C07280=1058.171,437.212,373.375,176.008,40.727,157.978
C07281=1058.182,437.458,373.325,176.019,40.739,157.981
C07282=1058.192,437.701,373.276,176.030,40.751,157.985
C07283=1058.202,437.947,373.225,176.042,40.763,157.989
C07284=1058.213,438.192,373.176,176.053,40.775,157.993
C07285=1058.223,438.436,373.126,176.064,40.788,157.997
C07286=1058.234,438.681,373.077,176.075,40.799,158.000
C07287=1058.244,438.926,373.026,176.086,40.811,158.004
C07288=1058.254,439.170,372.977,176.098,40.824,158.008
C07289=1058.265,439.415,372.926,176.109,40.836,158.012
C07290=1058.276,439.660,372.877,176.121,40.848,158.016
C07291=1058.286,439.904,372.826,176.133,40.860,158.020
C07292=1058.296,440.149,372.776,176.144,40.873,158.024
C07293=1058.307,440.394,372.725,176.155,40.885,158.028
C07294=1058.317,440.638,372.675,176.167,40.897,158.032
C07295=1058.328,440.882,372.625,176.179,40.909,158.035
C07296=1058.338,441.128,372.575,176.191,40.922,158.040
C07297=1058.349,441.372,372.525,176.202,40.935,158.044
C07298=1058.359,441.617,372.474,176.215,40.947,158.048
C07299=1058.370,441.861,372.423,176.226,40.960,158.052
C07300=1058.381,442.106,372.373,176.238,40.973,158.056
C07301=1058.391,442.350,372.322,176.250,40.985,158.060
C07302=1058.402,442.595,372.272,176.262,40.997,158.064
C07303=1058.414,442.840,372.220,176.274,41.010,158.068
C07304=1058.424,443.084,372.169,176.286,41.023,158.072
C07305=1058.435,443.329,372.118,176.299,41.036,158.076
C07306=1058.446,443.573,372.067,176.311,41.049,158.080
C07307=1058.456,443.817,372.017,176.323,41.062,158.085
C07308=1058.467,444.062,371.965,176.335,41.075,158.089
C07309=1058.479,444.330,371.909,176.349,41.089,158.094
C07310=1058.491,444.598,371.853,176.363,41.103,158.098
C07311=1058.503,444.866,371.797,176.377,41.117,158.103
C07312=1058.515,445.134,371.741,176.390,41.132,158.108
C07313=1058.525,445.378,371.690,176.403,41.145,158.112
C07314=1058.537,445.622,371.638,176.415,41.158,158.116
C07315=1058.548,445.867,371.587,176.428,41.171,158.121
C07316=1058.559,446.111,371.535,176.441,41.185,158.125
C07317=1058.570,446.355,371.484,176.454,41.198,158.129
C07318=1058.582,446.599,371.432,176.467,41.211,158.134
C07319=1058.592,446.842,371.380,176.480,41.225,158.138
C07320=1058.604,447.087,371.329,176.493,41.238,158.143
C07321=1058.616,447.330,371.279,176.506,41.251,158.147
C07322=1058.629,447.573,371.228,176.519,41.264,158.151
C07323=1058.642,447.817,371.178,176.532,41.277,158.156
C07324=1058.658,448.062,371.130,176.546,41.289,158.160
C07325=1058.673,448.306,371.080,176.558,41.302,158.164
C07326=1058.690,448.550,371.033,176.572,41.314,158.168
C07327=1058.707,448.795,370.986,176.586,41.325,158.172
C07328=1058.725,449.040,370.938,176.599,41.337,158.176
C07329=1058.744,449.285,370.893,176.613,41.348,158.180
C07330=1058.764,449.530,370.848,176.626,41.360,158.184
C07331=1058.785,449.776,370.802,176.641,41.371,158.188
C07332=1058.806,450.022,370.758,176.654,41.381,158.192
C07333=1058.477,450.035,370.476,176.650,41.491,158.222
C07334=1058.456,449.789,370.520,176.636,41.480,158.218
C07335=1058.436,449.544,370.565,176.622,41.470,158.214
C07336=1058.416,449.299,370.610,176.608,41.459,158.210
C07337=1058.396,449.054,370.656,176.594,41.447,158.206
C07338=1058.378,448.810,370.703,176.581,41.436,158.202
C07339=1058.361,448.565,370.750,176.567,41.424,158.198
C07340=1058.344,448.320,370.798,176.553,41.412,158.194
C07341=1058.328,448.076,370.847,176.540,41.400,158.190
C07342=1058.313,447.831,370.896,176.527,41.387,158.186
C07343=1058.299,447.587,370.945,176.514,41.375,158.182
C07344=1058.286,447.343,370.995,176.501,41.362,158.177
C07345=1058.273,447.100,371.046,176.487,41.349,158.173
C07346=1058.262,446.857,371.097,176.474,41.336,158.169
C07347=1058.251,446.613,371.149,176.461,41.322,158.164
C07348=1058.239,446.369,371.201,176.448,41.309,158.160
C07349=1058.229,446.124,371.252,176.435,41.295,158.155
C07350=1058.218,445.881,371.303,176.422,41.282,158.151
C07351=1058.206,445.636,371.355,176.409,41.269,158.147
C07352=1058.195,445.392,371.407,176.396,41.256,158.142
C07353=1058.184,445.147,371.459,176.384,41.243,158.138
C07354=1058.173,444.899,371.510,176.371,41.230,158.134
C07355=1058.162,444.651,371.563,176.359,41.217,158.129
C07356=1058.151,444.401,371.615,176.346,41.204,158.125
C07357=1058.139,444.153,371.667,176.333,41.190,158.121
C07358=1058.129,443.908,371.718,176.321,41.177,158.116
C07359=1058.117,443.664,371.769,176.308,41.164,158.112
C07360=1058.107,443.419,371.820,176.296,41.151,158.108
C07361=1058.096,443.175,371.872,176.283,41.139,158.104
C07362=1058.085,442.930,371.922,176.271,41.126,158.099
C07363=1058.075,442.686,371.974,176.259,41.113,158.095
C07364=1058.064,442.442,372.024,176.246,41.101,158.091
C07365=1058.054,442.197,372.075,176.235,41.088,158.087
C07366=1058.042,441.952,372.126,176.223,41.075,158.083
C07367=1058.031,441.707,372.176,176.211,41.063,158.079
C07368=1058.021,441.463,372.227,176.199,41.050,158.075
C07369=1058.010,441.218,372.277,176.186,41.038,158.071
C07370=1058.000,440.974,372.328,176.175,41.026,158.067
C07371=1057.989,440.729,372.379,176.163,41.013,158.063
C07372=1057.978,440.485,372.429,176.151,41.001,158.059
C07373=1057.968,440.240,372.479,176.139,40.988,158.055
C07374=1057.957,439.996,372.529,176.128,40.976,158.051
C07375=1057.947,439.751,372.579,176.117,40.964,158.047
C07376=1057.937,439.506,372.630,176.105,40.952,158.043
C07377=1057.926,439.261,372.680,176.093,40.940,158.039
C07378=1057.915,439.016,372.730,176.082,40.928,158.035
C07379=1057.905,438.772,372.780,176.070,40.915,158.031
C07380=1057.895,438.527,372.830,176.059,40.904,158.028
C07381=1057.884,438.282,372.879,176.048,40.892,158.024
C07382=1057.874,438.038,372.929,176.036,40.879,158.020
C07383=1057.864,437.793,372.980,176.025,40.867,158.016
C07384=1057.853,437.548,373.029,176.014,40.855,158.012
C07385=1057.843,437.304,373.078,176.003,40.844,158.009
C07386=1057.832,437.059,373.128,175.992,40.832,158.005
C07387=1057.822,436.814,373.178,175.981,40.820,158.001
C07388=1057.812,436.569,373.227,175.970,40.808,157.997
C07389=1057.801,436.324,373.276,175.959,40.797,157.994
C07390=1057.790,436.079,373.326,175.947,40.785,157.990
C07391=1057.780,435.834,373.375,175.936,40.774,157.986
C07392=1057.770,435.589,373.424,175.925,40.762,157.983
C07393=1057.760,435.345,373.473,175.915,40.751,157.979
C07394=1057.749,435.100,373.523,175.903,40.739,157.975
C07395=1057.739,434.855,373.572,175.893,40.727,157.972
C07396=1057.729,434.610,373.621,175.882,40.716,157.968
C07397=1057.719,434.365,373.670,175.872,40.705,157.965
C07398=1057.709,434.120,373.719,175.861,40.694,157.961
C07399=1057.699,433.875,373.767,175.851,40.682,157.958
C07400=1057.689,433.630,373.816,175.840,40.671,157.954
C07401=1057.679,433.385,373.866,175.829,40.660,157.951
C07402=1057.669,433.140,373.914,175.819,40.648,157.947
C07403=1057.658,432.895,373.963,175.809,40.637,157.944
C07404=1057.649,432.650,374.012,175.798,40.626,157.940
C07405=1057.639,432.405,374.061,175.788,40.615,157.937
C07406=1057.629,432.160,374.109,175.777,40.604,157.933
C07407=1057.619,431.915,374.158,175.767,40.593,157.930
C07408=1057.609,431.670,374.206,175.757,40.582,157.926
C07409=1057.600,431.425,374.255,175.746,40.571,157.923
C07410=1057.585,431.059,374.327,175.732,40.554,157.918
C07411=1057.571,430.692,374.399,175.716,40.538,157.913
C07412=1057.556,430.326,374.472,175.701,40.521,157.908
C07413=1057.541,429.960,374.544,175.686,40.505,157.903
C07414=1057.531,429.714,374.591,175.676,40.495,157.900
C07415=1057.522,429.469,374.640,175.666,40.484,157.896
C07416=1057.512,429.224,374.687,175.657,40.473,157.893
C07417=1057.502,428.979,374.736,175.646,40.462,157.890
C07418=1057.492,428.734,374.783,175.637,40.452,157.886
C07419=1057.482,428.489,374.831,175.627,40.441,157.883
C07420=1057.472,428.243,374.879,175.617,40.431,157.880
C07421=1057.463,427.998,374.927,175.607,40.420,157.877
C07422=1057.453,427.753,374.974,175.598,40.409,157.873
C07423=1057.444,427.508,375.022,175.587,40.399,157.870
C07424=1057.434,427.263,375.070,175.578,40.388,157.867
C07425=1057.424,427.017,375.117,175.569,40.378,157.864
C07426=1057.415,426.772,375.165,175.559,40.368,157.861
C07427=1057.406,426.527,375.213,175.550,40.357,157.858
C07428=1057.395,426.282,375.260,175.540,40.347,157.854
C07429=1057.386,426.036,375.308,175.530,40.337,157.851
C07430=1057.376,425.791,375.354,175.521,40.327,157.848
C07431=1057.367,425.545,375.402,175.512,40.316,157.845
C07432=1057.357,425.300,375.449,175.503,40.306,157.842
C07433=1057.348,425.055,375.496,175.493,40.296,157.839
C07434=1057.338,424.810,375.543,175.484,40.285,157.836
C07435=1057.329,424.564,375.590,175.475,40.276,157.833
C07436=1057.319,424.319,375.637,175.466,40.266,157.830
C07437=1057.309,424.073,375.684,175.457,40.256,157.827
C07438=1057.301,423.828,375.731,175.446,40.245,157.824
C07439=1057.291,423.582,375.778,175.437,40.236,157.821
C07440=1057.282,423.337,375.825,175.429,40.226,157.818
C07441=1057.272,423.091,375.872,175.420,40.215,157.815
C07442=1057.262,422.847,375.919,175.411,40.206,157.812
C07443=1057.254,422.601,375.965,175.402,40.196,157.809
C07444=1057.244,422.355,376.012,175.393,40.186,157.806
C07445=1057.235,422.110,376.059,175.384,40.176,157.803
C07446=1057.225,421.865,376.106,175.375,40.167,157.800
C07447=1057.216,421.619,376.152,175.365,40.156,157.797
C07448=1057.207,421.374,376.199,175.356,40.147,157.794
C07449=1057.197,421.128,376.245,175.347,40.137,157.791
C07450=1057.188,420.883,376.291,175.339,40.127,157.788
C07451=1057.180,420.637,376.338,175.330,40.117,157.785
C07452=1057.170,420.392,376.384,175.321,40.108,157.783
C07453=1057.161,420.146,376.431,175.313,40.099,157.780
C07454=1057.152,419.901,376.477,175.304,40.089,157.777
C07455=1057.143,419.655,376.523,175.296,40.079,157.774
C07456=1057.134,419.410,376.569,175.287,40.070,157.771
C07457=1057.124,419.164,376.615,175.278,40.060,157.768
C07458=1057.115,418.918,376.661,175.270,40.051,157.766
C07459=1057.105,418.673,376.707,175.261,40.041,157.763
C07460=1057.097,418.427,376.754,175.252,40.032,157.760
C07461=1057.088,418.181,376.799,175.243,40.023,157.757
C07462=1057.079,417.936,376.845,175.236,40.014,157.755
C07463=1057.070,417.690,376.891,175.227,40.004,157.752
C07464=1057.060,417.445,376.937,175.218,39.995,157.749
C07465=1057.051,417.199,376.983,175.210,39.985,157.746
C07466=1057.039,416.854,377.046,175.198,39.973,157.743
C07467=1057.025,416.509,377.111,175.186,39.960,157.739
C07468=1057.013,416.164,377.175,175.175,39.947,157.735
C07469=1057.001,415.819,377.239,175.164,39.934,157.731
C07470=1056.992,415.573,377.284,175.155,39.925,157.729
C07471=1056.983,415.327,377.330,175.147,39.916,157.726
C07472=1056.974,415.081,377.375,175.139,39.907,157.723
C07473=1056.965,414.836,377.420,175.131,39.897,157.721
C07474=1056.956,414.591,377.466,175.122,39.889,157.718
C07475=1056.947,414.345,377.511,175.115,39.880,157.716
C07476=1056.938,414.099,377.556,175.106,39.871,157.713
C07477=1056.929,413.853,377.602,175.098,39.862,157.710
C07478=1056.921,413.608,377.647,175.090,39.853,157.708
C07479=1056.912,413.362,377.692,175.082,39.844,157.705
C07480=1056.902,413.117,377.737,175.075,39.835,157.702
C07481=1056.894,412.870,377.782,175.066,39.826,157.700
C07482=1056.885,412.624,377.827,175.058,39.817,157.697
C07483=1056.876,412.378,377.872,175.050,39.809,157.695
C07484=1056.867,412.133,377.916,175.042,39.800,157.692
C07485=1056.858,411.887,377.962,175.035,39.791,157.690
C07486=1056.849,411.641,378.007,175.026,39.783,157.687
C07487=1056.840,411.396,378.051,175.019,39.774,157.685
C07488=1056.832,411.150,378.096,175.011,39.766,157.682
C07489=1056.823,410.903,378.140,175.004,39.757,157.680
C07490=1056.814,410.658,378.185,174.995,39.749,157.677
C07491=1056.805,410.412,378.230,174.988,39.740,157.675
C07492=1056.797,410.166,378.274,174.981,39.731,157.673
C07493=1056.787,409.921,378.319,174.973,39.723,157.670
C07494=1056.779,409.674,378.363,174.965,39.714,157.668
C07495=1056.771,409.428,378.408,174.957,39.705,157.665
C07496=1056.761,409.182,378.452,174.950,39.697,157.663
C07497=1056.753,408.936,378.496,174.942,39.689,157.660
C07498=1056.745,408.691,378.541,174.935,39.680,157.658
C07499=1056.735,408.445,378.585,174.927,39.672,157.656
C07500=1056.727,408.199,378.630,174.919,39.663,157.653
C07501=1056.719,407.953,378.674,174.912,39.655,157.651
C07502=1056.710,407.708,378.718,174.905,39.647,157.648
C07503=1056.702,407.462,378.763,174.897,39.638,157.646
C07504=1056.693,407.215,378.807,174.890,39.630,157.644
C07505=1056.685,406.969,378.850,174.883,39.622,157.641
C07506=1056.676,406.724,378.895,174.875,39.614,157.639
C07507=1056.667,406.477,378.939,174.868,39.605,157.637
C07508=1056.659,406.232,378.983,174.860,39.597,157.634
C07509=1056.651,405.986,379.027,174.852,39.589,157.632
C07510=1056.642,405.739,379.071,174.845,39.581,157.630
C07511=1056.634,405.493,379.115,174.838,39.573,157.627
C07512=1056.625,405.248,379.159,174.831,39.565,157.625
C07513=1056.617,405.002,379.202,174.823,39.556,157.623
C07514=1056.608,404.756,379.246,174.816,39.549,157.620
C07515=1056.600,404.509,379.290,174.809,39.540,157.618
C07516=1056.591,404.264,379.334,174.802,39.532,157.616
C07517=1056.583,404.018,379.377,174.794,39.525,157.614
C07518=1056.575,403.772,379.421,174.787,39.517,157.611
C07519=1056.566,403.526,379.464,174.781,39.508,157.609
C07520=1056.558,403.280,379.508,174.774,39.500,157.607
C07521=1056.550,403.034,379.552,174.767,39.493,157.605
C07522=1056.538,402.694,379.611,174.757,39.482,157.602
C07523=1056.526,402.355,379.671,174.747,39.471,157.599
C07524=1056.515,402.016,379.731,174.737,39.460,157.596
C07525=1056.503,401.678,379.791,174.728,39.450,157.593
C07526=1056.495,401.431,379.834,174.721,39.442,157.590
C07527=1056.487,401.185,379.877,174.714,39.434,157.588
C07528=1056.478,400.939,379.920,174.707,39.426,157.586
C07529=1056.470,400.693,379.963,174.700,39.419,157.584
C07530=1056.461,400.447,380.006,174.693,39.411,157.582
C07531=1056.453,400.201,380.049,174.687,39.403,157.580
C07532=1056.445,399.954,380.092,174.679,39.396,157.578
C07533=1056.437,399.708,380.135,174.672,39.388,157.575
C07534=1056.428,399.462,380.178,174.665,39.380,157.573
C07535=1056.420,399.216,380.221,174.658,39.373,157.571
C07536=1056.411,398.970,380.264,174.652,39.365,157.569
C07537=1056.403,398.724,380.307,174.645,39.358,157.567
C07538=1056.395,398.478,380.349,174.638,39.350,157.565
C07539=1056.387,398.232,380.392,174.631,39.342,157.563
C07540=1056.379,397.985,380.436,174.625,39.335,157.561
C07541=1056.371,397.739,380.478,174.618,39.328,157.559
C07542=1056.363,397.493,380.521,174.611,39.320,157.557
C07543=1056.355,397.247,380.563,174.605,39.313,157.555
C07544=1056.346,397.001,380.606,174.599,39.306,157.553
C07545=1056.339,396.755,380.648,174.592,39.298,157.550
C07546=1056.330,396.509,380.691,174.585,39.291,157.548
C07547=1056.322,396.262,380.734,174.579,39.283,157.546
C07548=1056.313,396.016,380.777,174.572,39.276,157.544
C07549=1056.305,395.770,380.818,174.565,39.269,157.542
C07550=1056.297,395.523,380.860,174.559,39.261,157.540
C07551=1056.288,395.277,380.903,174.552,39.254,157.538
C07552=1056.281,395.031,380.945,174.545,39.247,157.536
C07553=1056.272,394.785,380.988,174.539,39.239,157.534
C07554=1056.265,394.539,381.029,174.532,39.232,157.532
C07555=1056.256,394.293,381.072,174.527,39.225,157.530
C07556=1056.249,394.047,381.114,174.520,39.218,157.528
C07557=1056.241,393.800,381.157,174.513,39.211,157.526
C07558=1056.232,393.554,381.198,174.507,39.204,157.524
C07559=1056.224,393.308,381.240,174.500,39.197,157.523
C07560=1056.216,393.062,381.282,174.494,39.189,157.520
C07561=1056.208,392.815,381.325,174.487,39.182,157.519
C07562=1056.201,392.569,381.367,174.481,39.175,157.517
C07563=1056.192,392.323,381.408,174.475,39.168,157.515
C07564=1056.184,392.077,381.450,174.468,39.161,157.513
C07565=1056.176,391.830,381.493,174.462,39.154,157.511
C07566=1056.168,391.584,381.535,174.455,39.147,157.509
C07567=1056.160,391.338,381.576,174.450,39.140,157.507
C07568=1056.152,391.091,381.617,174.443,39.133,157.505
C07569=1056.145,390.845,381.659,174.437,39.126,157.503
C07570=1056.136,390.599,381.701,174.430,39.119,157.501
C07571=1056.128,390.353,381.743,174.425,39.112,157.499
C07572=1056.121,390.106,381.784,174.418,39.105,157.498
C07573=1056.112,389.861,381.826,174.412,39.098,157.496
C07574=1056.104,389.614,381.868,174.405,39.092,157.494
C07575=1056.097,389.367,381.909,174.400,39.085,157.492
C07576=1056.088,389.121,381.951,174.393,39.078,157.490
C07577=1056.080,388.875,381.992,174.387,39.071,157.488
C07578=1056.070,388.553,382.046,174.379,39.062,157.486
C07579=1056.059,388.231,382.100,174.371,39.054,157.484
C07580=1056.049,387.910,382.154,174.364,39.045,157.481
C07581=1056.039,387.589,382.207,174.356,39.036,157.479
C07582=1056.030,387.342,382.248,174.349,39.029,157.477
C07583=1056.023,387.096,382.290,174.343,39.023,157.475
C07584=1056.015,386.849,382.331,174.337,39.016,157.473
C07585=1056.007,386.603,382.372,174.331,39.010,157.472
C07586=1055.999,386.357,382.413,174.325,39.003,157.470
C07587=1055.990,386.110,382.454,174.319,38.996,157.468
C07588=1055.983,385.864,382.496,174.313,38.989,157.466
C07589=1055.975,385.617,382.536,174.307,38.983,157.464
C07590=1055.968,385.371,382.578,174.301,38.977,157.463
C07591=1055.960,385.124,382.618,174.295,38.970,157.461
C07592=1055.952,384.878,382.659,174.289,38.963,157.459
C07593=1055.944,384.632,382.700,174.283,38.957,157.457
C07594=1055.936,384.385,382.741,174.277,38.950,157.456
C07595=1055.929,384.139,382.782,174.272,38.944,157.454
C07596=1055.921,383.892,382.822,174.266,38.937,157.452
C07597=1055.913,383.646,382.863,174.259,38.931,157.450
C07598=1055.906,383.400,382.904,174.254,38.924,157.449
C07599=1055.898,383.153,382.945,174.248,38.918,157.447
C07600=1055.890,382.906,382.985,174.242,38.911,157.445
C07601=1055.883,382.660,383.026,174.236,38.905,157.443
C07602=1055.875,382.413,383.067,174.231,38.898,157.442
C07603=1055.867,382.167,383.108,174.225,38.892,157.440
C07604=1055.859,381.921,383.149,174.219,38.886,157.438
C07605=1055.852,381.674,383.189,174.213,38.879,157.437
C07606=1055.844,381.427,383.230,174.208,38.873,157.435
C07607=1055.836,381.181,383.270,174.202,38.867,157.433
C07608=1055.829,380.934,383.310,174.197,38.860,157.432
C07609=1055.822,380.688,383.351,174.190,38.854,157.430
C07610=1055.814,380.441,383.391,174.184,38.847,157.428
C07611=1055.806,380.195,383.432,174.179,38.842,157.427
C07612=1055.799,379.948,383.472,174.173,38.835,157.425
C07613=1055.791,379.702,383.512,174.168,38.829,157.423
C07614=1055.783,379.455,383.552,174.162,38.823,157.422
C07615=1055.775,379.208,383.592,174.156,38.817,157.420
C07616=1055.767,378.962,383.633,174.151,38.810,157.418
C07617=1055.760,378.715,383.672,174.145,38.804,157.417
C07618=1055.752,378.468,383.712,174.140,38.798,157.415
C07619=1055.744,378.222,383.753,174.134,38.792,157.414
C07620=1055.736,377.975,383.793,174.129,38.786,157.412
C07621=1055.729,377.728,383.833,174.122,38.780,157.410
C07622=1055.722,377.482,383.872,174.117,38.774,157.409
C07623=1055.714,377.236,383.913,174.112,38.768,157.407
C07624=1055.706,376.989,383.953,174.106,38.761,157.405
C07625=1055.698,376.742,383.993,174.101,38.755,157.404
C07626=1055.691,376.496,384.032,174.095,38.750,157.402
C07627=1055.683,376.249,384.072,174.090,38.744,157.401
C07628=1055.676,376.002,384.112,174.084,38.737,157.399
C07629=1055.668,375.756,384.152,174.079,38.731,157.397
C07630=1055.661,375.509,384.192,174.074,38.725,157.396
C07631=1055.653,375.262,384.232,174.067,38.719,157.394
C07632=1055.646,375.016,384.271,174.062,38.713,157.393
C07633=1055.638,374.769,384.311,174.056,38.708,157.391
C07634=1055.630,374.479,384.357,174.051,38.700,157.389
C07635=1055.621,374.189,384.404,174.044,38.693,157.388
C07636=1055.611,373.900,384.451,174.038,38.686,157.386
C07637=1055.603,373.610,384.497,174.031,38.679,157.384
C07638=1055.596,373.363,384.537,174.026,38.673,157.382
C07639=1055.589,373.116,384.576,174.020,38.668,157.381
C07640=1055.581,372.869,384.616,174.015,38.662,157.379
C07641=1055.574,372.623,384.656,174.011,38.656,157.378
C07642=1055.567,372.376,384.695,174.005,38.650,157.376
C07643=1055.559,372.130,384.734,174.000,38.644,157.375
C07644=1055.552,371.883,384.774,173.995,38.638,157.373
C07645=1055.544,371.636,384.813,173.989,38.633,157.372
C07646=1055.536,371.389,384.853,173.984,38.627,157.370
C07647=1055.530,371.142,384.891,173.979,38.622,157.369
C07648=1055.521,370.896,384.931,173.973,38.616,157.367
C07649=1055.514,370.649,384.970,173.968,38.610,157.366
C07650=1055.506,370.402,385.009,173.963,38.604,157.364
C07651=1055.499,370.156,385.048,173.958,38.599,157.363
C07652=1055.492,369.908,385.087,173.952,38.593,157.361
C07653=1055.484,369.662,385.126,173.947,38.587,157.360
C07654=1055.476,369.415,385.165,173.942,38.581,157.358
C07655=1055.470,369.168,385.204,173.936,38.576,157.357
C07656=1055.462,368.922,385.243,173.931,38.570,157.355
C07657=1055.454,368.674,385.282,173.926,38.565,157.354
C07658=1055.447,368.428,385.320,173.921,38.559,157.353
C07659=1055.440,368.181,385.359,173.916,38.553,157.351
C07660=1055.432,367.934,385.399,173.911,38.548,157.350
C07661=1055.425,367.688,385.437,173.906,38.542,157.348
C07662=1055.418,367.441,385.476,173.901,38.537,157.347
C07663=1055.410,367.194,385.515,173.895,38.531,157.345
C07664=1055.403,366.947,385.554,173.890,38.526,157.344
C07665=1055.396,366.700,385.592,173.885,38.520,157.342
C07666=1055.389,366.474,385.628,173.881,38.515,157.341
C07667=1055.383,366.248,385.663,173.876,38.510,157.340
C07668=1055.375,366.022,385.699,173.871,38.505,157.339
C07669=1055.369,365.796,385.735,173.866,38.500,157.337
C07670=1055.362,365.570,385.770,173.862,38.494,157.336
C07671=1055.355,365.344,385.806,173.857,38.490,157.335
C07672=1055.349,365.118,385.840,173.853,38.485,157.333
C07673=1055.342,364.892,385.876,173.848,38.480,157.332
C07674=1055.335,364.645,385.914,173.843,38.474,157.331
C07675=1055.328,364.397,385.953,173.839,38.469,157.329
C07676=1055.320,364.151,385.991,173.833,38.463,157.328
C07677=1055.313,363.904,386.030,173.828,38.458,157.326
C07678=1055.306,363.657,386.068,173.823,38.453,157.325
C07679=1055.299,363.411,386.107,173.819,38.447,157.324
C07680=1055.292,363.163,386.145,173.814,38.442,157.322
C07681=1055.284,362.916,386.183,173.808,38.436,157.321
C07682=1055.277,362.669,386.222,173.803,38.431,157.320
C07683=1055.270,362.422,386.260,173.798,38.426,157.318
C07684=1055.262,362.176,386.298,173.794,38.420,157.317
C07685=1055.256,361.928,386.336,173.789,38.415,157.315
C07686=1055.248,361.682,386.374,173.784,38.410,157.314
C07687=1055.241,361.435,386.412,173.779,38.405,157.313
C07688=1055.234,361.188,386.451,173.774,38.399,157.311
C07689=1055.226,360.941,386.489,173.769,38.394,157.310
C07690=1055.217,360.628,386.537,173.763,38.387,157.308
C07691=1055.208,360.316,386.585,173.757,38.380,157.307
C07692=1055.199,360.002,386.633,173.751,38.374,157.305
C07693=1055.189,359.689,386.681,173.744,38.367,157.303
C07694=1055.182,359.442,386.720,173.739,38.362,157.302
C07695=1055.175,359.195,386.757,173.735,38.357,157.301
C07696=1055.168,358.948,386.795,173.730,38.352,157.299
C07697=1055.160,358.702,386.833,173.725,38.347,157.298
C07698=1055.153,358.454,386.870,173.721,38.342,157.297
C07699=1055.147,358.207,386.908,173.716,38.336,157.295
C07700=1055.139,357.960,386.946,173.711,38.331,157.294
C07701=1055.132,357.713,386.984,173.707,38.326,157.293
C07702=1055.125,357.466,387.022,173.702,38.321,157.291
C07703=1055.118,357.220,387.059,173.697,38.316,157.290
C07704=1055.111,356.973,387.096,173.692,38.311,157.289
C07705=1055.103,356.725,387.134,173.687,38.305,157.288
C07706=1055.096,356.478,387.171,173.682,38.301,157.286
C07707=1055.089,356.231,387.209,173.678,38.296,157.285
C07708=1055.082,355.984,387.247,173.673,38.291,157.284
C07709=1055.074,355.737,387.284,173.669,38.285,157.282
C07710=1055.067,355.490,387.322,173.664,38.280,157.281
C07711=1055.060,355.243,387.359,173.659,38.275,157.280
C07712=1055.053,354.996,387.397,173.655,38.270,157.279
C07713=1055.045,354.748,387.434,173.650,38.265,157.277
C07714=1055.039,354.502,387.471,173.646,38.260,157.276
C07715=1055.032,354.255,387.509,173.641,38.255,157.275
C07716=1055.024,354.008,387.546,173.636,38.251,157.274
C07717=1055.017,353.761,387.584,173.632,38.245,157.272
C07718=1055.010,353.513,387.621,173.627,38.240,157.271
C07719=1055.003,353.266,387.658,173.623,38.235,157.270
C07720=1054.996,353.019,387.695,173.618,38.230,157.269
C07721=1054.989,352.772,387.733,173.614,38.225,157.267
C07722=1054.982,352.524,387.770,173.608,38.220,157.266
C07723=1054.975,352.278,387.807,173.603,38.215,157.265
C07724=1054.968,352.031,387.844,173.599,38.210,157.264
C07725=1054.961,351.783,387.881,173.595,38.206,157.263
C07726=1054.954,351.536,387.919,173.590,38.201,157.261
C07727=1054.947,351.289,387.956,173.585,38.196,157.260
C07728=1054.940,351.042,387.993,173.581,38.191,157.259
C07729=1054.933,350.795,388.030,173.576,38.186,157.258
C07730=1054.926,350.548,388.066,173.572,38.181,157.256
C07731=1054.919,350.301,388.104,173.567,38.177,157.255
C07732=1054.912,350.053,388.140,173.563,38.172,157.254
C07733=1054.905,349.806,388.178,173.558,38.167,157.253
C07734=1054.898,349.559,388.214,173.554,38.162,157.251
C07735=1054.890,349.312,388.251,173.550,38.157,157.250
C07736=1054.883,349.064,388.288,173.546,38.152,157.249
C07737=1054.877,348.817,388.325,173.541,38.147,157.248
C07738=1054.869,348.570,388.362,173.537,38.143,157.247
C07739=1054.862,348.322,388.398,173.532,38.138,157.246
C07740=1054.856,348.075,388.435,173.528,38.133,157.244
C07741=1054.849,347.828,388.472,173.523,38.129,157.243
C07742=1054.842,347.582,388.508,173.519,38.124,157.242
C07743=1054.835,347.334,388.545,173.515,38.119,157.241
C07744=1054.828,347.087,388.582,173.510,38.114,157.240
C07745=1054.820,346.840,388.618,173.506,38.109,157.238
C07746=1054.813,346.574,388.657,173.501,38.104,157.237
C07747=1054.805,346.307,388.697,173.496,38.099,157.236
C07748=1054.798,346.041,388.736,173.492,38.094,157.235
C07749=1054.790,345.775,388.776,173.487,38.089,157.233
C07750=1054.784,345.528,388.813,173.482,38.084,157.232
C07751=1054.776,345.280,388.849,173.478,38.080,157.231
C07752=1054.770,345.033,388.885,173.474,38.075,157.230
C07753=1054.762,344.786,388.922,173.469,38.071,157.229
C07754=1054.756,344.539,388.958,173.465,38.066,157.228
C07755=1054.749,344.291,388.995,173.460,38.061,157.226
C07756=1054.742,344.044,389.031,173.456,38.057,157.225
C07757=1054.735,343.797,389.067,173.452,38.052,157.224
C07758=1054.728,343.550,389.103,173.447,38.047,157.223
C07759=1054.721,343.303,389.140,173.444,38.043,157.222
C07760=1054.714,343.055,389.177,173.440,38.038,157.221
C07761=1054.708,342.808,389.212,173.435,38.033,157.220
C07762=1054.700,342.560,389.248,173.431,38.029,157.219
C07763=1054.694,342.313,389.285,173.426,38.025,157.217
C07764=1054.686,342.066,389.321,173.422,38.020,157.216
C07765=1054.680,341.819,389.357,173.418,38.015,157.215
C07766=1054.673,341.571,389.392,173.413,38.011,157.214
C07767=1054.665,341.324,389.429,173.409,38.006,157.213
C07768=1054.659,341.077,389.465,173.405,38.002,157.212
C07769=1054.652,340.829,389.500,173.401,37.997,157.211
C07770=1054.644,340.582,389.536,173.397,37.993,157.210
C07771=1054.638,340.335,389.573,173.393,37.988,157.209
C07772=1054.631,340.087,389.608,173.388,37.984,157.207
C07773=1054.624,339.840,389.645,173.384,37.980,157.206
C07774=1054.617,339.593,389.681,173.380,37.975,157.205
C07775=1054.610,339.345,389.716,173.375,37.970,157.204
C07776=1054.604,339.098,389.753,173.371,37.966,157.203
C07777=1054.597,338.851,389.788,173.367,37.961,157.202
C07778=1054.589,338.603,389.824,173.364,37.957,157.201
C07779=1054.583,338.355,389.860,173.359,37.952,157.200
C07780=1054.576,338.109,389.895,173.355,37.948,157.199
C07781=1054.569,337.861,389.931,173.351,37.943,157.198
C07782=1054.562,337.614,389.967,173.346,37.939,157.196
C07783=1054.556,337.366,390.003,173.342,37.934,157.195
C07784=1054.549,337.120,390.038,173.338,37.930,157.194
C07785=1054.542,336.872,390.074,173.335,37.925,157.193
C07786=1054.536,336.624,390.109,173.330,37.922,157.192
C07787=1054.528,336.377,390.145,173.326,37.917,157.191
C07788=1054.521,336.130,390.181,173.322,37.913,157.190
C07789=1054.515,335.882,390.216,173.318,37.908,157.189
C07790=1054.508,335.635,390.251,173.313,37.904,157.188
C07791=1054.500,335.387,390.287,173.310,37.899,157.187
C07792=1054.494,335.140,390.323,173.306,37.895,157.186
C07793=1054.487,334.892,390.358,173.302,37.891,157.185
C07794=1054.481,334.645,390.393,173.298,37.886,157.184
C07795=1054.474,334.398,390.428,173.293,37.882,157.183
C07796=1054.466,334.150,390.464,173.290,37.878,157.182
C07797=1054.459,333.903,390.500,173.286,37.874,157.181
C07798=1054.453,333.656,390.535,173.282,37.869,157.179
C07799=1054.446,333.408,390.570,173.277,37.865,157.178
C07800=1054.439,333.161,390.605,173.273,37.861,157.177
C07801=1054.432,332.913,390.640,173.269,37.856,157.176
C07802=1054.425,332.643,390.679,173.266,37.852,157.175
C07803=1054.418,332.372,390.717,173.261,37.847,157.174
C07804=1054.410,332.103,390.756,173.257,37.842,157.173
C07805=1054.402,331.832,390.794,173.252,37.838,157.172
C07806=1054.396,331.585,390.829,173.248,37.833,157.171
C07807=1054.389,331.337,390.865,173.244,37.829,157.170
C07808=1054.382,331.090,390.900,173.240,37.825,157.169
C07809=1054.375,330.843,390.935,173.237,37.820,157.168
C07810=1054.369,330.595,390.969,173.232,37.817,157.167
C07811=1054.362,330.347,391.004,173.228,37.812,157.166
C07812=1054.355,330.100,391.039,173.224,37.808,157.165
C07813=1054.349,329.853,391.075,173.220,37.804,157.164
C07814=1054.342,329.605,391.110,173.217,37.800,157.163
C07815=1054.335,329.357,391.144,173.213,37.795,157.162
C07816=1054.328,329.110,391.179,173.208,37.791,157.161
C07817=1054.320,328.862,391.214,173.204,37.787,157.160
C07818=1054.314,328.614,391.249,173.201,37.783,157.159
C07819=1054.306,328.367,391.283,173.197,37.779,157.158
C07820=1054.300,328.120,391.318,173.193,37.775,157.157
C07821=1054.293,327.872,391.353,173.189,37.771,157.156
C07822=1054.286,327.625,391.387,173.186,37.767,157.155
C07823=1054.279,327.377,391.422,173.182,37.763,157.154
C07824=1054.272,327.130,391.456,173.177,37.758,157.153
C07825=1054.265,326.882,391.491,173.173,37.754,157.152
C07826=1054.259,326.634,391.526,173.170,37.750,157.151
C07827=1054.252,326.388,391.560,173.166,37.746,157.150
C07828=1054.245,326.140,391.594,173.162,37.742,157.149
C07829=1054.238,325.893,391.630,173.158,37.738,157.148
C07830=1054.231,325.645,391.663,173.155,37.734,157.147
C07831=1054.224,325.398,391.698,173.151,37.730,157.146
C07832=1054.218,325.150,391.733,173.147,37.726,157.145
C07833=1054.211,324.902,391.767,173.143,37.722,157.144
C07834=1054.204,324.655,391.802,173.140,37.718,157.143
C07835=1054.197,324.407,391.836,173.135,37.714,157.142
C07836=1054.190,324.160,391.871,173.131,37.710,157.141
C07837=1054.184,323.912,391.905,173.127,37.705,157.140
C07838=1054.177,323.665,391.939,173.124,37.701,157.139
C07839=1054.170,323.417,391.974,173.120,37.697,157.138
C07840=1054.163,323.170,392.008,173.116,37.694,157.137
C07841=1054.157,322.922,392.042,173.113,37.690,157.136
C07842=1054.150,322.674,392.076,173.109,37.686,157.135
C07843=1054.143,322.427,392.111,173.105,37.682,157.134
C07844=1054.137,322.179,392.145,173.101,37.677,157.133
C07845=1054.129,321.932,392.179,173.098,37.673,157.132
C07846=1054.123,321.684,392.213,173.094,37.669,157.131
C07847=1054.116,321.437,392.248,173.090,37.665,157.131
C07848=1054.110,321.189,392.282,173.086,37.661,157.130
C07849=1054.103,320.941,392.316,173.083,37.657,157.129
C07850=1054.096,320.694,392.350,173.079,37.653,157.128
C07851=1054.090,320.446,392.384,173.075,37.650,157.127
C07852=1054.083,320.199,392.418,173.072,37.646,157.126
C07853=1054.076,319.951,392.452,173.068,37.642,157.125
C07854=1054.070,319.704,392.486,173.064,37.637,157.124
C07855=1054.063,319.456,392.520,173.060,37.633,157.123
C07856=1054.056,319.208,392.554,173.057,37.629,157.122
C07857=1054.050,318.961,392.588,173.053,37.625,157.121
C07858=1054.042,318.685,392.627,173.049,37.621,157.120
C07859=1054.035,318.410,392.664,173.046,37.617,157.119
C07860=1054.027,318.134,392.702,173.041,37.612,157.118
C07861=1054.020,317.859,392.740,173.037,37.608,157.117
C07862=1054.014,317.611,392.774,173.033,37.604,157.116
C07863=1054.007,317.364,392.808,173.030,37.600,157.115
C07864=1054.001,317.116,392.842,173.026,37.596,157.114
C07865=1053.994,316.869,392.875,173.022,37.592,157.113
C07866=1053.988,316.621,392.910,173.019,37.588,157.112
C07867=1053.982,316.373,392.943,173.016,37.584,157.111
C07868=1053.975,316.125,392.977,173.012,37.580,157.110
C07869=1053.968,315.878,393.011,173.008,37.576,157.109
C07870=1053.962,315.630,393.045,173.005,37.572,157.108
C07871=1053.955,315.382,393.079,173.001,37.568,157.108
C07872=1053.949,315.135,393.113,172.997,37.564,157.107
C07873=1053.943,314.888,393.146,172.994,37.560,157.106
C07874=1053.936,314.640,393.180,172.990,37.556,157.105
C07875=1053.930,314.393,393.213,172.987,37.553,157.104
C07876=1053.923,314.144,393.247,172.984,37.549,157.103
C07877=1053.917,313.897,393.281,172.980,37.545,157.102
C07878=1053.910,313.649,393.315,172.976,37.541,157.101
C07879=1053.904,313.402,393.348,172.973,37.537,157.100
C07880=1053.897,313.154,393.382,172.969,37.533,157.099
C07881=1053.890,312.907,393.415,172.965,37.529,157.098
C07882=1053.883,312.658,393.448,172.962,37.525,157.098
C07883=1053.877,312.412,393.482,172.958,37.522,157.097
C07884=1053.870,312.163,393.515,172.955,37.518,157.096
C07885=1053.863,311.916,393.548,172.952,37.514,157.095
C07886=1053.856,311.668,393.581,172.948,37.510,157.094
C07887=1053.850,311.420,393.614,172.944,37.507,157.093
C07888=1053.843,311.173,393.648,172.941,37.503,157.092
C07889=1053.837,310.925,393.681,172.937,37.499,157.091
C07890=1053.829,310.677,393.714,172.933,37.495,157.090
C07891=1053.823,310.430,393.747,172.930,37.491,157.090
C07892=1053.816,310.182,393.780,172.927,37.488,157.089
C07893=1053.810,309.935,393.814,172.923,37.484,157.088
C07894=1053.803,309.686,393.847,172.920,37.481,157.087
C07895=1053.796,309.439,393.880,172.916,37.477,157.086
C07896=1053.788,309.191,393.913,172.913,37.473,157.085
C07897=1053.782,308.944,393.946,172.909,37.469,157.084
C07898=1053.776,308.696,393.978,172.905,37.465,157.083
C07899=1053.769,308.448,394.011,172.903,37.462,157.083
C07900=1053.762,308.201,394.045,172.899,37.458,157.082
C07901=1053.756,307.953,394.078,172.895,37.454,157.081
C07902=1053.749,307.705,394.111,172.892,37.450,157.080
C07903=1053.743,307.457,394.143,172.888,37.447,157.079
C07904=1053.736,307.210,394.177,172.885,37.443,157.078
C07905=1053.729,306.962,394.210,172.882,37.440,157.078
C07906=1053.722,306.715,394.242,172.878,37.436,157.077
C07907=1053.716,306.467,394.275,172.875,37.432,157.076
C07908=1053.709,306.219,394.308,172.871,37.428,157.075
C07909=1053.703,305.971,394.341,172.868,37.425,157.074
C07910=1053.697,305.724,394.374,172.865,37.421,157.073
C07911=1053.690,305.475,394.407,172.861,37.417,157.072
C07912=1053.683,305.228,394.439,172.858,37.413,157.071
C07913=1053.676,304.981,394.472,172.854,37.410,157.071
C07914=1053.669,304.709,394.508,172.850,37.406,157.070
C07915=1053.662,304.438,394.544,172.847,37.402,157.069
C07916=1053.655,304.166,394.580,172.843,37.397,157.068
C07917=1053.648,303.896,394.615,172.839,37.393,157.067
C07918=1053.641,303.647,394.649,172.837,37.390,157.066
C07919=1053.635,303.400,394.681,172.833,37.386,157.065
C07920=1053.628,303.152,394.714,172.829,37.382,157.064
C07921=1053.622,302.905,394.747,172.826,37.379,157.064
C07922=1053.616,302.657,394.779,172.823,37.375,157.063
C07923=1053.608,302.408,394.811,172.820,37.372,157.062
C07924=1053.602,302.161,394.844,172.816,37.368,157.061
C07925=1053.596,301.913,394.877,172.812,37.364,157.060
C07926=1053.590,301.666,394.910,172.810,37.360,157.059
C07927=1053.583,301.418,394.942,172.806,37.357,157.058
C07928=1053.576,301.171,394.974,172.802,37.353,157.057
C07929=1053.570,300.923,395.006,172.800,37.349,157.057
C07930=1053.563,300.674,395.040,172.796,37.346,157.056
C07931=1053.557,300.427,395.072,172.793,37.342,157.055
C07932=1053.551,300.179,395.105,172.790,37.338,157.054
C07933=1053.544,299.932,395.137,172.786,37.334,157.053
C07934=1053.538,299.684,395.169,172.783,37.331,157.052
C07935=1053.531,299.436,395.202,172.780,37.328,157.052
C07936=1053.525,299.188,395.235,172.777,37.324,157.051
C07937=1053.519,298.940,395.267,172.773,37.320,157.050
C07938=1053.512,298.693,395.299,172.770,37.316,157.049
C07939=1053.506,298.445,395.332,172.767,37.313,157.048
C07940=1053.500,298.197,395.364,172.763,37.309,157.047
C07941=1053.494,297.950,395.396,172.761,37.305,157.047
C07942=1053.488,297.701,395.428,172.757,37.302,157.046
C07943=1053.481,297.454,395.461,172.753,37.298,157.045
C07944=1053.474,297.206,395.493,172.751,37.294,157.044
C07945=1053.468,296.958,395.525,172.747,37.291,157.043
C07946=1053.462,296.711,395.558,172.744,37.287,157.042
C07947=1053.455,296.463,395.589,172.741,37.283,157.042
C07948=1053.449,296.215,395.622,172.738,37.280,157.041
C07949=1053.442,295.967,395.654,172.734,37.276,157.040
C07950=1053.436,295.720,395.686,172.731,37.272,157.039
C07951=1053.429,295.472,395.718,172.728,37.269,157.038
C07952=1053.423,295.224,395.750,172.725,37.266,157.038
C07953=1053.416,294.976,395.782,172.722,37.262,157.037
C07954=1053.410,294.727,395.814,172.718,37.258,157.036
C07955=1053.403,294.479,395.846,172.716,37.255,157.035
C07956=1053.397,294.232,395.879,172.712,37.251,157.034
C07957=1053.390,293.984,395.910,172.708,37.248,157.033
C07958=1053.384,293.736,395.942,172.706,37.244,157.033
C07959=1053.377,293.488,395.974,172.702,37.241,157.032
C07960=1053.371,293.241,396.005,172.700,37.237,157.031
C07961=1053.365,292.993,396.037,172.696,37.233,157.030
C07962=1053.358,292.745,396.069,172.693,37.230,157.029
C07963=1053.351,292.498,396.101,172.690,37.226,157.029
C07964=1053.345,292.250,396.133,172.687,37.223,157.028
C07965=1053.338,292.002,396.164,172.684,37.219,157.027
C07966=1053.332,291.754,396.196,172.680,37.216,157.026
C07967=1053.326,291.506,396.228,172.677,37.213,157.025
C07968=1053.319,291.258,396.259,172.674,37.209,157.025
C07969=1053.312,291.010,396.291,172.671,37.205,157.024
C07970=1053.306,290.755,396.325,172.668,37.202,157.023
C07971=1053.299,290.499,396.357,172.665,37.198,157.022
C07972=1053.293,290.244,396.389,172.661,37.195,157.021
C07973=1053.286,289.988,396.422,172.658,37.191,157.021
C07974=1053.279,289.740,396.453,172.655,37.187,157.020
C07975=1053.272,289.493,396.485,172.652,37.184,157.019
C07976=1053.266,289.244,396.517,172.649,37.180,157.018
C07977=1053.260,288.996,396.548,172.645,37.177,157.017
C07978=1053.253,288.749,396.579,172.643,37.173,157.017
C07979=1053.247,288.501,396.611,172.639,37.170,157.016
C07980=1053.241,288.253,396.643,172.637,37.166,157.015
C07981=1053.234,288.005,396.674,172.633,37.163,157.014
C07982=1053.227,287.757,396.706,172.631,37.159,157.014
C07983=1053.221,287.509,396.736,172.627,37.156,157.013
C07984=1053.214,287.261,396.768,172.625,37.153,157.012
C07985=1053.208,287.014,396.799,172.621,37.149,157.011
C07986=1053.201,286.766,396.830,172.618,37.146,157.010
C07987=1053.195,286.518,396.862,172.615,37.142,157.010
C07988=1053.188,286.270,396.893,172.612,37.139,157.009
C07989=1053.181,286.021,396.924,172.609,37.135,157.008
C07990=1053.175,285.773,396.956,172.606,37.132,157.007
C07991=1053.169,285.526,396.987,172.603,37.128,157.006
C07992=1053.163,285.278,397.018,172.600,37.125,157.006
C07993=1053.156,285.030,397.049,172.597,37.121,157.005
C07994=1053.149,284.782,397.080,172.594,37.118,157.004
C07995=1053.143,284.534,397.112,172.591,37.114,157.003
C07996=1053.137,284.287,397.143,172.588,37.111,157.003
C07997=1053.130,284.038,397.174,172.585,37.107,157.002
C07998=1053.123,283.790,397.205,172.582,37.104,157.001
C07999=1053.117,283.542,397.237,172.579,37.100,157.000
C08000=1053.111,283.294,397.267,172.576,37.097,156.999
C08001=1053.104,283.047,397.298,172.572,37.094,156.999
C08002=1053.098,282.798,397.329,172.570,37.090,156.998
C08003=1053.091,282.550,397.360,172.567,37.087,156.997
C08004=1053.085,282.303,397.392,172.564,37.084,156.997
C08005=1053.078,282.054,397.422,172.560,37.080,156.996
C08006=1053.072,281.806,397.454,172.558,37.077,156.995
C08007=1053.066,281.559,397.484,172.554,37.073,156.994
C08008=1053.059,281.311,397.515,172.552,37.070,156.993
C08009=1053.053,281.062,397.546,172.549,37.066,156.993
C08010=1053.047,280.815,397.577,172.546,37.063,156.992
C08011=1053.040,280.567,397.608,172.543,37.059,156.991
C08012=1053.034,280.319,397.639,172.540,37.056,156.990
C08013=1053.028,280.071,397.670,172.537,37.052,156.990
C08014=1053.021,279.823,397.701,172.534,37.049,156.989
C08015=1053.015,279.574,397.732,172.531,37.045,156.988
C08016=1053.009,279.327,397.762,172.529,37.042,156.987
C08017=1053.002,279.079,397.794,172.525,37.039,156.987
C08018=1052.995,278.830,397.824,172.523,37.036,156.986
C08019=1052.989,278.583,397.855,172.519,37.032,156.985
C08020=1052.982,278.335,397.886,172.517,37.029,156.984
C08021=1052.976,278.086,397.916,172.514,37.025,156.983
C08022=1052.970,277.840,397.946,172.511,37.022,156.983
C08023=1052.963,277.594,397.977,172.508,37.019,156.982
C08024=1052.957,277.348,398.007,172.505,37.015,156.981
C08025=1052.951,277.102,398.037,172.502,37.012,156.980
C08026=1052.944,276.857,398.068,172.500,37.008,156.980
C08027=1052.938,276.610,398.098,172.496,37.005,156.979
C08028=1052.931,276.364,398.128,172.494,37.002,156.978
C08029=1052.925,276.118,398.159,172.490,36.998,156.978
C08030=1052.918,275.870,398.190,172.488,36.995,156.977
C08031=1052.912,275.622,398.221,172.485,36.991,156.976
C08032=1052.905,275.374,398.250,172.482,36.988,156.975
C08033=1052.899,275.126,398.281,172.479,36.985,156.975
C08034=1052.893,274.878,398.312,172.477,36.981,156.974
C08035=1052.886,274.630,398.342,172.473,36.978,156.973
C08036=1052.880,274.382,398.372,172.471,36.974,156.972
C08037=1052.874,274.133,398.403,172.468,36.971,156.971
C08038=1052.866,273.886,398.434,172.465,36.968,156.971
C08039=1052.861,273.638,398.464,172.462,36.965,156.970
C08040=1052.854,273.389,398.495,172.459,36.961,156.969
C08041=1052.848,273.142,398.524,172.456,36.958,156.969
C08042=1052.841,272.893,398.555,172.454,36.954,156.968
C08043=1052.835,272.645,398.585,172.450,36.951,156.967
C08044=1052.828,272.397,398.616,172.448,36.948,156.966
C08045=1052.822,272.149,398.646,172.445,36.944,156.966
C08046=1052.816,271.901,398.677,172.442,36.941,156.965
C08047=1052.809,271.653,398.706,172.439,36.937,156.964
C08048=1052.803,271.404,398.736,172.437,36.934,156.963
C08049=1052.797,271.157,398.766,172.433,36.931,156.963
C08050=1052.790,270.908,398.797,172.431,36.927,156.962
C08051=1052.784,270.661,398.827,172.428,36.924,156.961
C08052=1052.777,270.412,398.857,172.426,36.921,156.960
C08053=1052.771,270.165,398.887,172.422,36.917,156.960
C08054=1052.764,269.916,398.918,172.420,36.914,156.959
C08055=1052.758,269.668,398.947,172.418,36.911,156.958
C08056=1052.752,269.420,398.977,172.414,36.907,156.957
C08057=1052.745,269.172,399.007,172.412,36.904,156.957
C08058=1052.739,268.924,399.038,172.409,36.900,156.956
C08059=1052.732,268.676,399.068,172.406,36.897,156.955
C08060=1052.727,268.428,399.097,172.403,36.894,156.955
C08061=1052.719,268.179,399.128,172.401,36.890,156.954
C08062=1052.713,267.932,399.157,172.398,36.887,156.953
C08063=1052.707,267.683,399.187,172.395,36.884,156.952
C08064=1052.700,267.435,399.217,172.392,36.880,156.952
C08065=1052.694,267.187,399.247,172.390,36.877,156.951
C08066=1052.688,266.938,399.277,172.386,36.874,156.950
C08067=1052.681,266.691,399.307,172.384,36.871,156.949
C08068=1052.675,266.442,399.337,172.381,36.867,156.949
C08069=1052.668,266.194,399.366,172.379,36.864,156.948
C08070=1052.662,265.947,399.396,172.375,36.861,156.947
C08071=1052.655,265.698,399.427,172.373,36.857,156.946
C08072=1052.649,265.450,399.456,172.370,36.854,156.946
C08073=1052.643,265.203,399.486,172.368,36.851,156.945
C08074=1052.636,264.953,399.516,172.364,36.847,156.944
C08075=1052.630,264.706,399.545,172.362,36.844,156.944
C08076=1052.624,264.458,399.574,172.360,36.841,156.943
C08077=1052.617,264.209,399.605,172.357,36.837,156.942
C08078=1052.610,263.966,399.634,172.354,36.834,156.941
C08079=1052.605,263.721,399.663,172.351,36.831,156.941
C08080=1052.598,263.478,399.692,172.349,36.827,156.940
C08081=1052.592,263.234,399.722,172.346,36.824,156.939
C08082=1052.587,262.989,399.751,172.344,36.821,156.939
C08083=1052.579,262.745,399.780,172.341,36.817,156.938
C08084=1052.573,262.501,399.809,172.338,36.814,156.937
C08085=1052.566,262.257,399.837,172.335,36.811,156.936
C08086=1052.560,262.009,399.867,172.333,36.808,156.936
C08087=1052.553,261.761,399.897,172.330,36.804,156.935
C08088=1052.547,261.513,399.926,172.327,36.801,156.934
C08089=1052.540,261.264,399.955,172.325,36.798,156.934
C08090=1052.534,261.016,399.984,172.322,36.795,156.933
C08091=1052.527,260.768,400.014,172.320,36.791,156.932
C08092=1052.520,260.520,400.043,172.317,36.788,156.932
C08093=1052.514,260.271,400.072,172.314,36.785,156.931
C08094=1052.508,260.023,400.101,172.311,36.782,156.930
C08095=1052.501,259.776,400.131,172.309,36.778,156.929
C08096=1052.494,259.527,400.161,172.306,36.775,156.929
C08097=1052.488,259.279,400.190,172.304,36.772,156.928
C08098=1052.482,259.031,400.219,172.301,36.768,156.927
C08099=1052.475,258.782,400.248,172.298,36.766,156.927
C08100=1052.468,258.534,400.278,172.296,36.762,156.926
C08101=1052.462,258.286,400.307,172.293,36.759,156.925
C08102=1052.456,258.038,400.336,172.291,36.756,156.924
C08103=1052.449,257.789,400.365,172.287,36.752,156.924
C08104=1052.443,257.541,400.394,172.285,36.749,156.923
C08105=1052.437,257.293,400.423,172.282,36.746,156.922
C08106=1052.430,257.045,400.452,172.280,36.743,156.922
C08107=1052.423,256.796,400.481,172.278,36.739,156.921
C08108=1052.417,256.548,400.510,172.275,36.736,156.920
C08109=1052.410,256.300,400.539,172.272,36.733,156.920
C08110=1052.404,256.052,400.568,172.269,36.729,156.919
C08111=1052.397,255.804,400.598,172.267,36.726,156.918
C08112=1052.391,255.556,400.628,172.264,36.723,156.917
C08113=1052.384,255.307,400.657,172.262,36.720,156.917
C08114=1052.378,255.059,400.686,172.259,36.716,156.916
C08115=1052.372,254.811,400.715,172.257,36.713,156.915
C08116=1052.366,254.562,400.743,172.254,36.710,156.915
C08117=1052.360,254.314,400.772,172.251,36.706,156.914
C08118=1052.353,254.065,400.801,172.249,36.703,156.913
C08119=1052.347,253.817,400.830,172.246,36.700,156.912
C08120=1052.340,253.569,400.859,172.244,36.696,156.912
C08121=1052.333,253.321,400.888,172.241,36.693,156.911
C08122=1052.327,253.073,400.917,172.239,36.690,156.910
C08123=1052.321,252.825,400.946,172.237,36.687,156.910
C08124=1052.315,252.577,400.975,172.234,36.683,156.909
C08125=1052.308,252.329,401.004,172.231,36.680,156.908
C08126=1052.302,252.080,401.032,172.228,36.677,156.907
C08127=1052.296,251.831,401.062,172.226,36.673,156.907
C08128=1052.289,251.583,401.091,172.223,36.670,156.906
C08129=1052.282,251.335,401.119,172.221,36.667,156.905
C08130=1052.276,251.087,401.148,172.218,36.663,156.905
C08131=1052.270,250.839,401.177,172.216,36.660,156.904
C08132=1052.264,250.590,401.206,172.214,36.657,156.903
C08133=1052.258,250.342,401.235,172.211,36.653,156.902
C08134=1052.252,250.098,401.264,172.209,36.650,156.902
C08135=1052.245,249.852,401.291,172.206,36.647,156.901
C08136=1052.239,249.608,401.320,172.204,36.644,156.900
C08137=1052.233,249.362,401.349,172.201,36.640,156.900
C08138=1052.227,249.118,401.377,172.199,36.636,156.899
C08139=1052.220,248.872,401.405,172.196,36.634,156.898
C08140=1052.215,248.628,401.434,172.194,36.630,156.898
C08141=1052.208,248.382,401.462,172.192,36.627,156.897
C08142=1052.202,248.134,401.491,172.189,36.623,156.896
C08143=1052.196,247.885,401.519,172.187,36.620,156.895
C08144=1052.190,247.638,401.548,172.184,36.617,156.895
C08145=1052.184,247.390,401.577,172.182,36.613,156.894
C08146=1052.177,247.141,401.605,172.179,36.610,156.893
C08147=1052.171,246.893,401.634,172.177,36.607,156.893
C08148=1052.165,246.645,401.662,172.175,36.603,156.892
C08149=1052.159,246.396,401.691,172.172,36.600,156.891
C08150=1052.152,246.148,401.720,172.170,36.596,156.890
C08151=1052.146,245.900,401.748,172.167,36.593,156.890
C08152=1052.139,245.652,401.777,172.165,36.590,156.889
C08153=1052.133,245.403,401.805,172.162,36.587,156.888
C08154=1052.126,245.155,401.834,172.159,36.583,156.888
C08155=1052.121,244.906,401.862,172.156,36.580,156.887
C08156=1052.114,244.658,401.891,172.154,36.577,156.886
C08157=1052.108,244.410,401.919,172.152,36.573,156.885
C08158=1052.102,244.161,401.947,172.149,36.570,156.885
C08159=1052.095,243.913,401.975,172.147,36.567,156.884
C08160=1052.089,243.665,402.004,172.144,36.563,156.883
C08161=1052.082,243.416,402.033,172.142,36.560,156.883
C08162=1052.076,243.168,402.061,172.141,36.557,156.882
C08163=1052.070,242.920,402.088,172.138,36.554,156.881
C08164=1052.063,242.672,402.117,172.136,36.550,156.881
C08165=1052.058,242.423,402.145,172.133,36.547,156.880
C08166=1052.051,242.175,402.173,172.131,36.544,156.879
C08167=1052.045,241.927,402.202,172.128,36.540,156.878
C08168=1052.039,241.678,402.230,172.126,36.536,156.878
C08169=1052.032,241.430,402.258,172.124,36.533,156.877
C08170=1052.025,241.182,402.287,172.121,36.530,156.876
C08171=1052.019,240.933,402.315,172.119,36.527,156.876
C08172=1052.012,240.685,402.343,172.116,36.523,156.875
C08173=1052.006,240.436,402.370,172.114,36.520,156.874
C08174=1052.000,240.188,402.398,172.111,36.517,156.874
C08175=1051.993,239.940,402.427,172.109,36.514,156.873
C08176=1051.987,239.691,402.455,172.107,36.510,156.872
C08177=1051.981,239.443,402.483,172.104,36.507,156.872
C08178=1051.974,239.195,402.511,172.102,36.504,156.871
C08179=1051.968,238.946,402.539,172.099,36.500,156.870
C08180=1051.961,238.697,402.567,172.097,36.497,156.869
C08181=1051.955,238.449,402.594,172.095,36.494,156.869
C08182=1051.949,238.202,402.623,172.092,36.491,156.868
C08183=1051.942,237.953,402.651,172.090,36.487,156.867
C08184=1051.936,237.705,402.678,172.087,36.484,156.867
C08185=1051.929,237.456,402.706,172.085,36.481,156.866
C08186=1051.923,237.207,402.734,172.083,36.478,156.865
C08187=1051.916,236.959,402.762,172.081,36.474,156.864
C08188=1051.910,236.711,402.790,172.079,36.471,156.864
C08189=1051.904,236.463,402.818,172.076,36.468,156.863
C08190=1051.898,236.214,402.846,172.074,36.464,156.862
C08191=1051.891,235.967,402.874,172.072,36.461,156.862
C08192=1051.885,235.719,402.901,172.069,36.457,156.861
C08193=1051.879,235.471,402.929,172.067,36.455,156.860
C08194=1051.872,235.223,402.956,172.064,36.451,156.860
C08195=1051.866,234.975,402.984,172.062,36.447,156.859
C08196=1051.859,234.728,403.012,172.059,36.444,156.858
C08197=1051.853,234.479,403.040,172.058,36.441,156.858
C08198=1051.847,234.230,403.068,172.056,36.438,156.857
C08199=1051.841,233.983,403.095,172.053,36.434,156.856
C08200=1051.834,233.734,403.122,172.051,36.431,156.855
C08201=1051.828,233.485,403.150,172.048,36.428,156.855
C08202=1051.822,233.236,403.178,172.046,36.424,156.854
C08203=1051.816,232.989,403.206,172.044,36.421,156.853
C08204=1051.809,232.740,403.234,172.041,36.418,156.853
C08205=1051.802,232.492,403.261,172.040,36.414,156.852
C08206=1051.796,232.244,403.289,172.037,36.411,156.851
C08207=1051.790,231.995,403.316,172.035,36.407,156.851
C08208=1051.784,231.746,403.344,172.033,36.405,156.850
C08209=1051.777,231.498,403.372,172.030,36.401,156.849
C08210=1051.771,231.250,403.399,172.028,36.397,156.848
C08211=1051.765,231.001,403.426,172.025,36.394,156.848
C08212=1051.758,230.752,403.454,172.023,36.391,156.847
C08213=1051.752,230.505,403.481,172.022,36.388,156.846
C08214=1051.745,230.256,403.509,172.019,36.384,156.846
C08215=1051.739,230.007,403.536,172.017,36.381,156.845
C08216=1051.733,229.759,403.563,172.014,36.378,156.844
C08217=1051.727,229.511,403.592,172.012,36.374,156.844
C08218=1051.721,229.262,403.619,172.010,36.371,156.843
C08219=1051.714,229.014,403.646,172.008,36.368,156.842
C08220=1051.708,228.765,403.674,172.006,36.364,156.841
C08221=1051.701,228.517,403.700,172.003,36.361,156.841
C08222=1051.694,228.268,403.728,172.001,36.357,156.840
C08223=1051.688,228.021,403.755,171.999,36.354,156.839
C08224=1051.682,227.772,403.782,171.996,36.351,156.839
C08225=1051.675,227.523,403.810,171.995,36.348,156.838
C08226=1051.669,227.275,403.837,171.992,36.344,156.837
C08227=1051.662,227.026,403.864,171.990,36.341,156.837
C08228=1051.656,226.777,403.891,171.988,36.338,156.836
C08229=1051.650,226.529,403.919,171.985,36.334,156.835
C08230=1051.643,226.281,403.945,171.984,36.331,156.835
C08231=1051.636,226.032,403.973,171.981,36.328,156.834
C08232=1051.630,225.784,404.000,171.979,36.325,156.833
C08233=1051.624,225.535,404.027,171.977,36.321,156.832
C08234=1051.618,225.287,404.054,171.974,36.317,156.832
C08235=1051.611,225.039,404.082,171.973,36.314,156.831
C08236=1051.605,224.790,404.109,171.970,36.311,156.830
C08237=1051.599,224.542,404.136,171.968,36.307,156.830
C08238=1051.592,224.293,404.162,171.966,36.304,156.829
C08239=1051.586,224.045,404.190,171.963,36.301,156.828
C08240=1051.579,223.796,404.217,171.962,36.298,156.828
C08241=1051.573,223.547,404.244,171.959,36.294,156.827
C08242=1051.567,223.300,404.271,171.957,36.291,156.826
C08243=1051.560,223.050,404.298,171.955,36.288,156.826
C08244=1051.555,222.802,404.325,171.953,36.284,156.825
C08245=1051.547,222.554,404.352,171.951,36.280,156.824
C08246=1051.541,222.306,404.379,171.949,36.277,156.823
C08247=1051.535,222.057,404.406,171.946,36.274,156.823
C08248=1051.529,221.809,404.433,171.945,36.270,156.822
C08249=1051.523,221.560,404.460,171.942,36.267,156.821
C08250=1051.516,221.305,404.488,171.940,36.264,156.821
C08251=1051.509,221.050,404.515,171.938,36.260,156.820
C08252=1051.503,220.794,404.543,171.935,36.256,156.819
C08253=1051.496,220.540,404.570,171.934,36.253,156.818
C08254=1051.490,220.291,404.597,171.931,36.250,156.818
C08255=1051.484,220.043,404.624,171.929,36.246,156.817
C08256=1051.477,219.794,404.651,171.927,36.243,156.816
C08257=1051.471,219.546,404.678,171.925,36.240,156.816
C08258=1051.464,219.297,404.704,171.923,36.237,156.815
C08259=1051.458,219.049,404.731,171.920,36.233,156.814
C08260=1051.452,218.800,404.758,171.918,36.230,156.814
C08261=1051.445,218.552,404.784,171.917,36.227,156.813
C08262=1051.438,218.303,404.811,171.914,36.223,156.812
C08263=1051.432,218.055,404.838,171.912,36.220,156.812
C08264=1051.426,217.806,404.865,171.911,36.216,156.811
C08265=1051.420,217.558,404.891,171.908,36.213,156.810
C08266=1051.413,217.309,404.918,171.906,36.210,156.809
C08267=1051.407,217.061,404.944,171.903,36.206,156.809
C08268=1051.400,216.812,404.971,171.902,36.203,156.808
C08269=1051.394,216.564,404.997,171.900,36.200,156.807
C08270=1051.387,216.315,405.024,171.897,36.196,156.807
C08271=1051.381,216.067,405.050,171.896,36.192,156.806
C08272=1051.375,215.818,405.077,171.893,36.189,156.805
C08273=1051.368,215.569,405.103,171.891,36.186,156.805
C08274=1051.362,215.320,405.130,171.890,36.182,156.804
C08275=1051.355,215.072,405.157,171.887,36.179,156.803
C08276=1051.350,214.824,405.183,171.885,36.176,156.802
C08277=1051.342,214.575,405.210,171.884,36.172,156.802
C08278=1051.337,214.327,405.236,171.881,36.169,156.801
C08279=1051.330,214.078,405.263,171.879,36.165,156.800
C08280=1051.324,213.830,405.289,171.877,36.162,156.800
C08281=1051.317,213.582,405.315,171.875,36.159,156.799
C08282=1051.311,213.333,405.342,171.873,36.155,156.798
C08283=1051.305,213.084,405.369,171.871,36.152,156.798
C08284=1051.299,212.836,405.395,171.869,36.148,156.797
C08285=1051.292,212.587,405.422,171.867,36.145,156.796
C08286=1051.286,212.339,405.448,171.865,36.141,156.795
C08287=1051.279,212.090,405.475,171.863,36.138,156.795
C08288=1051.273,211.841,405.501,171.860,36.134,156.794
C08289=1051.267,211.593,405.527,171.859,36.131,156.793
C08290=1051.260,211.344,405.554,171.857,36.128,156.793
C08291=1051.254,211.096,405.580,171.854,36.124,156.792
C08292=1051.248,210.848,405.606,171.853,36.121,156.791
C08293=1051.241,210.599,405.632,171.850,36.117,156.791
C08294=1051.235,210.350,405.658,171.848,36.114,156.790
C08295=1051.229,210.102,405.685,171.847,36.111,156.789
C08296=1051.222,209.853,405.711,171.844,36.107,156.788
C08297=1051.215,209.605,405.737,171.843,36.104,156.788
C08298=1051.209,209.356,405.763,171.841,36.100,156.787
C08299=1051.203,209.108,405.790,171.838,36.097,156.786
C08300=1051.196,208.860,405.816,171.837,36.093,156.786
C08301=1051.190,208.610,405.842,171.834,36.090,156.785
C08302=1051.184,208.362,405.868,171.832,36.087,156.784
C08303=1051.177,208.114,405.894,171.831,36.083,156.784
C08304=1051.171,207.865,405.919,171.828,36.080,156.783
C08305=1051.164,207.616,405.946,171.827,36.076,156.782
C08306=1051.158,207.367,405.972,171.825,36.073,156.781
C08307=1051.152,207.117,405.998,171.822,36.069,156.781
C08308=1051.145,206.868,406.024,171.821,36.066,156.780
C08309=1051.139,206.618,406.050,171.819,36.063,156.779
C08310=1051.113,205.566,406.156,171.593,35.967,156.761
C08311=1051.107,205.318,406.182,171.591,35.964,156.760
C08312=1051.101,205.068,406.206,171.588,35.962,156.760
C08313=1051.095,204.820,406.231,171.585,35.959,156.759
C08314=1051.089,204.572,406.257,171.583,35.956,156.759
C08315=1051.083,204.322,406.281,171.581,35.954,156.758
C08316=1051.077,204.074,406.307,171.577,35.952,156.758
C08317=1051.070,203.826,406.331,171.575,35.948,156.757
C08318=1051.064,203.577,406.356,171.573,35.946,156.757
C08319=1051.058,203.328,406.381,171.571,35.944,156.756
C08320=1051.052,203.079,406.406,171.567,35.941,156.756
C08321=1051.047,202.831,406.431,171.565,35.938,156.755
C08322=1051.041,202.582,406.456,171.563,35.936,156.755
C08323=1051.035,202.333,406.481,171.561,35.933,156.754
C08324=1051.029,202.085,406.506,171.557,35.930,156.754
C08325=1051.023,201.836,406.530,171.555,35.928,156.753
C08326=1051.017,201.587,406.556,171.553,35.925,156.753
C08327=1051.010,201.338,406.580,171.551,35.923,156.752
C08328=1051.005,201.090,406.605,171.547,35.920,156.752
C08329=1050.998,200.841,406.629,171.545,35.917,156.751
C08330=1050.992,200.592,406.654,171.543,35.915,156.751
C08331=1050.986,200.343,406.679,171.541,35.912,156.750
C08332=1050.980,200.095,406.702,171.537,35.910,156.750
C08333=1050.974,199.846,406.728,171.535,35.908,156.749
C08334=1050.967,199.597,406.752,171.533,35.905,156.749
C08335=1050.961,199.349,406.777,171.531,35.903,156.748
C08336=1050.956,199.100,406.801,171.527,35.900,156.748
C08337=1050.949,198.851,406.825,171.525,35.898,156.747
C08338=1050.943,198.602,406.850,171.523,35.895,156.747
C08339=1050.937,198.354,406.874,171.521,35.893,156.746
C08340=1050.931,198.105,406.899,171.517,35.890,156.746
C08341=1050.924,197.856,406.924,171.515,35.888,156.745
C08342=1050.919,197.608,406.948,171.513,35.886,156.745
C08343=1050.913,197.358,406.972,171.511,35.883,156.744
C08344=1050.906,197.110,406.997,171.507,35.881,156.744
C08345=1050.900,196.861,407.021,171.505,35.878,156.743
C08346=1050.894,196.612,407.045,171.503,35.875,156.743
C08347=1050.888,196.364,407.070,171.501,35.873,156.742
C08348=1050.882,196.116,407.094,171.498,35.870,156.742
C08349=1050.876,195.866,407.119,171.495,35.868,156.741
C08350=1050.870,195.618,407.143,171.493,35.865,156.741
C08351=1050.864,195.369,407.167,171.491,35.863,156.740
C08352=1050.858,195.121,407.192,171.488,35.860,156.740
C08353=1050.851,194.872,407.216,171.486,35.858,156.740
C08354=1050.846,194.622,407.241,171.483,35.855,156.739
C08355=1050.840,194.374,407.265,171.481,35.853,156.739
C08356=1050.834,194.125,407.289,171.479,35.851,156.738
C08357=1050.828,193.877,407.313,171.476,35.848,156.738
C08358=1050.821,193.628,407.338,171.474,35.846,156.737
C08359=1050.815,193.380,407.362,171.471,35.843,156.737
C08360=1050.809,193.130,407.387,171.469,35.841,156.736
C08361=1050.803,192.882,407.410,171.466,35.838,156.736
C08362=1050.798,192.633,407.435,171.464,35.836,156.735
C08363=1050.791,192.384,407.459,171.462,35.833,156.735
C08364=1050.786,192.135,407.483,171.460,35.831,156.734
C08365=1050.780,191.886,407.508,171.456,35.828,156.734
C08366=1050.774,191.638,407.531,171.454,35.826,156.733
C08367=1050.768,191.388,407.556,171.452,35.824,156.733
C08368=1050.762,191.140,407.580,171.450,35.821,156.732
C08369=1050.756,190.891,407.604,171.447,35.819,156.732
C08370=1050.750,190.643,407.628,171.445,35.816,156.731
C08371=1050.740,190.248,407.667,171.441,35.813,156.731
C08372=1050.731,189.854,407.705,171.438,35.809,156.730
C08373=1050.721,189.458,407.743,171.434,35.805,156.729
C08374=1050.712,189.064,407.782,171.430,35.801,156.728
C08375=1050.706,188.815,407.805,171.428,35.798,156.728
C08376=1050.700,188.565,407.829,171.425,35.796,156.727
C08377=1050.694,188.317,407.853,171.423,35.793,156.727
C08378=1050.689,188.069,407.877,171.421,35.791,156.727
C08379=1050.682,187.820,407.901,171.419,35.789,156.726
C08380=1050.677,187.571,407.926,171.415,35.786,156.726
C08381=1050.670,187.322,407.950,171.413,35.784,156.725
C08382=1050.665,187.073,407.974,171.411,35.781,156.725
C08383=1050.659,186.825,407.998,171.409,35.779,156.724
C08384=1050.653,186.575,408.021,171.407,35.777,156.724
C08385=1050.647,186.327,408.045,171.404,35.774,156.723
C08386=1050.642,186.078,408.069,171.402,35.772,156.723
C08387=1050.635,185.829,408.093,171.400,35.769,156.722
C08388=1050.629,185.581,408.117,171.398,35.767,156.722
C08389=1050.624,185.331,408.141,171.395,35.765,156.721
C08390=1050.618,185.083,408.165,171.393,35.762,156.721
C08391=1050.612,184.834,408.189,171.390,35.760,156.720
C08392=1050.606,184.585,408.213,171.388,35.757,156.720
C08393=1050.600,184.337,408.237,171.385,35.755,156.719
C08394=1050.595,184.088,408.260,171.383,35.752,156.719
C08395=1050.585,183.701,408.297,171.380,35.749,156.718
C08396=1050.575,183.313,408.334,171.377,35.745,156.718
C08397=1050.566,182.927,408.370,171.372,35.742,156.717
C08398=1050.556,182.539,408.407,171.369,35.738,156.716
C08399=1050.550,182.290,408.431,171.367,35.736,156.716
C08400=1050.543,182.042,408.453,171.365,35.734,156.715
C08401=1050.537,181.793,408.477,171.362,35.732,156.715
C08402=1050.531,181.544,408.500,171.360,35.729,156.715
C08403=1050.525,181.295,408.524,171.358,35.727,156.714
C08404=1050.518,181.046,408.548,171.355,35.725,156.714
C08405=1050.513,180.798,408.571,171.353,35.723,156.713
C08406=1050.507,180.549,408.595,171.350,35.720,156.713
C08407=1050.500,180.300,408.618,171.348,35.718,156.712
C08408=1050.494,180.051,408.641,171.346,35.716,156.712
C08409=1050.488,179.803,408.664,171.344,35.714,156.712
C08410=1050.482,179.553,408.688,171.342,35.711,156.711
C08411=1050.476,179.305,408.711,171.339,35.709,156.711
C08412=1050.470,179.056,408.734,171.337,35.707,156.710
C08413=1050.463,178.807,408.758,171.335,35.705,156.710
C08414=1050.457,178.558,408.781,171.333,35.702,156.709
C08415=1050.451,178.310,408.804,171.331,35.700,156.709
C08416=1050.445,178.060,408.828,171.328,35.698,156.709
C08417=1050.439,177.811,408.851,171.326,35.696,156.708
C08418=1050.433,177.563,408.874,171.323,35.694,156.708
C08419=1050.427,177.314,408.898,171.321,35.691,156.707
C08420=1050.421,177.065,408.921,171.319,35.689,156.707
C08421=1050.415,176.816,408.944,171.316,35.687,156.706
C08422=1050.409,176.567,408.967,171.314,35.685,156.706
C08423=1050.402,176.319,408.991,171.312,35.682,156.706
C08424=1050.396,176.070,409.014,171.310,35.680,156.705
C08425=1050.390,175.821,409.036,171.308,35.678,156.705
C08426=1050.385,175.572,409.059,171.305,35.676,156.704
C08427=1050.378,175.323,409.083,171.303,35.674,156.704
C08428=1050.372,175.074,409.106,171.301,35.671,156.703
C08429=1050.367,174.825,409.129,171.299,35.669,156.703
C08430=1050.361,174.577,409.153,171.297,35.667,156.703
C08431=1050.353,174.292,409.179,171.294,35.664,156.702
C08432=1050.347,174.007,409.205,171.291,35.662,156.702
C08433=1050.339,173.723,409.232,171.289,35.659,156.701
C08434=1050.333,173.438,409.258,171.287,35.656,156.701
C08435=1050.327,173.189,409.281,171.285,35.655,156.700
C08436=1050.320,172.940,409.305,171.282,35.652,156.700
C08437=1050.314,172.691,409.328,171.280,35.650,156.699
C08438=1050.308,172.442,409.351,171.278,35.648,156.699
C08439=1050.303,172.194,409.374,171.276,35.645,156.699
C08440=1050.297,171.945,409.397,171.274,35.643,156.698
C08441=1050.291,171.696,409.419,171.271,35.641,156.698
C08442=1050.284,171.447,409.443,171.269,35.639,156.697
C08443=1050.278,171.198,409.466,171.267,35.637,156.697
C08444=1050.272,170.949,409.489,171.265,35.635,156.697
C08445=1050.267,170.700,409.512,171.263,35.632,156.696
C08446=1050.261,170.452,409.535,171.260,35.630,156.696
C08447=1050.255,170.203,409.558,171.258,35.628,156.695
C08448=1050.249,169.954,409.581,171.256,35.625,156.695
C08449=1050.242,169.704,409.603,171.254,35.624,156.694
C08450=1050.237,169.456,409.626,171.252,35.621,156.694
C08451=1050.231,169.207,409.649,171.249,35.619,156.693
C08452=1050.225,168.958,409.672,171.247,35.617,156.693
C08453=1050.219,168.710,409.696,171.245,35.614,156.693
C08454=1050.213,168.461,409.718,171.243,35.612,156.692
C08455=1050.207,168.212,409.741,171.241,35.610,156.692
C08456=1050.201,167.963,409.764,171.238,35.608,156.691
C08457=1050.195,167.714,409.787,171.236,35.606,156.691
C08458=1050.190,167.465,409.810,171.234,35.603,156.691
C08459=1050.183,167.217,409.832,171.232,35.601,156.690
C08460=1050.178,166.968,409.855,171.230,35.599,156.690
C08461=1050.172,166.719,409.878,171.228,35.597,156.689
C08462=1050.166,166.469,409.900,171.226,35.594,156.689
C08463=1050.161,166.221,409.923,171.224,35.592,156.689
C08464=1050.154,165.971,409.946,171.222,35.590,156.688
C08465=1050.148,165.722,409.969,171.220,35.588,156.688
C08466=1050.142,165.473,409.992,171.218,35.586,156.687
C08467=1050.136,165.225,410.015,171.215,35.583,156.687
C08468=1050.131,164.976,410.038,171.213,35.581,156.686
C08469=1050.124,164.727,410.060,171.211,35.579,156.686
C08470=1050.118,164.478,410.083,171.209,35.577,156.686
C08471=1050.113,164.229,410.106,171.207,35.574,156.685
C08472=1050.107,163.980,410.129,171.204,35.572,156.685
C08473=1050.102,163.732,410.151,171.202,35.570,156.684
C08474=1050.096,163.483,410.173,171.200,35.568,156.684
C08475=1050.090,163.234,410.196,171.199,35.566,156.683
C08476=1050.084,162.985,410.219,171.197,35.563,156.683
C08477=1050.079,162.736,410.242,171.195,35.561,156.683
C08478=1050.072,162.487,410.264,171.192,35.559,156.682
C08479=1050.067,162.238,410.287,171.190,35.556,156.682
C08480=1050.061,161.989,410.310,171.188,35.555,156.681
C08481=1050.055,161.740,410.333,171.186,35.552,156.681
C08482=1050.049,161.492,410.355,171.184,35.550,156.681
C08483=1050.043,161.242,410.377,171.181,35.548,156.680
C08484=1050.038,160.993,410.400,171.179,35.546,156.680
C08485=1050.032,160.745,410.423,171.178,35.543,156.679
C08486=1050.026,160.495,410.445,171.176,35.541,156.679
C08487=1050.020,160.246,410.468,171.174,35.539,156.678
C08488=1050.013,159.998,410.490,171.172,35.537,156.678
C08489=1050.007,159.749,410.512,171.169,35.535,156.678
C08490=1050.002,159.500,410.535,171.167,35.533,156.677
C08491=1049.995,159.251,410.557,171.165,35.531,156.677
C08492=1049.990,159.002,410.579,171.163,35.528,156.676
C08493=1049.983,158.753,410.601,171.161,35.527,156.676
C08494=1049.977,158.504,410.623,171.158,35.525,156.676
C08495=1049.971,158.219,410.649,171.156,35.522,156.675
C08496=1049.964,157.933,410.675,171.154,35.520,156.675
C08497=1049.957,157.649,410.700,171.152,35.517,156.674
C08498=1049.950,157.364,410.725,171.150,35.515,156.674
C08499=1049.944,157.115,410.748,171.148,35.513,156.674
C08500=1049.938,156.866,410.770,171.145,35.511,156.673
C08501=1049.932,156.617,410.792,171.143,35.508,156.673
C08502=1049.926,156.368,410.814,171.141,35.507,156.672
C08503=1049.920,156.119,410.837,171.139,35.505,156.672
C08504=1049.914,155.870,410.859,171.137,35.502,156.672
C08505=1049.907,155.621,410.881,171.136,35.500,156.671
C08506=1049.902,155.372,410.903,171.133,35.498,156.671
C08507=1049.895,155.123,410.925,171.131,35.496,156.670
C08508=1049.890,154.875,410.947,171.129,35.494,156.670
C08509=1049.884,154.626,410.970,171.127,35.492,156.670
C08510=1049.878,154.376,410.991,171.125,35.490,156.669
C08511=1049.872,154.127,411.013,171.123,35.488,156.669
C08512=1049.865,153.879,411.035,171.120,35.486,156.669
C08513=1049.860,153.629,411.058,171.119,35.483,156.668
C08514=1049.854,153.381,411.080,171.117,35.482,156.668
C08515=1049.847,153.131,411.102,171.115,35.480,156.667
C08516=1049.841,152.882,411.123,171.113,35.477,156.667
C08517=1049.835,152.634,411.145,171.111,35.475,156.667
C08518=1049.830,152.385,411.167,171.108,35.473,156.666
C08519=1049.824,152.136,411.189,171.106,35.471,156.666
C08520=1049.817,151.887,411.211,171.104,35.469,156.665
C08521=1049.811,151.638,411.233,171.103,35.467,156.665
C08522=1049.806,151.388,411.255,171.101,35.465,156.665
C08523=1049.799,151.140,411.278,171.099,35.463,156.664
C08524=1049.794,150.891,411.299,171.096,35.461,156.664
C08525=1049.787,150.642,411.320,171.094,35.459,156.664
C08526=1049.781,150.393,411.342,171.092,35.457,156.663
C08527=1049.776,150.144,411.365,171.091,35.455,156.663
C08528=1049.769,149.895,411.387,171.089,35.453,156.662
C08529=1049.764,149.646,411.408,171.087,35.451,156.662
C08530=1049.758,149.397,411.430,171.084,35.448,156.662
C08531=1049.751,149.148,411.452,171.082,35.447,156.661
C08532=1049.745,148.899,411.474,171.080,35.445,156.661
C08533=1049.739,148.650,411.495,171.078,35.442,156.660
C08534=1049.734,148.401,411.517,171.077,35.440,156.660
C08535=1049.728,148.152,411.539,171.075,35.438,156.660
C08536=1049.721,147.903,411.561,171.072,35.437,156.659
C08537=1049.715,147.654,411.583,171.070,35.434,156.659
C08538=1049.709,147.405,411.604,171.068,35.432,156.659
C08539=1049.704,147.156,411.626,171.067,35.430,156.658
C08540=1049.697,146.907,411.647,171.065,35.428,156.658
C08541=1049.691,146.658,411.669,171.063,35.426,156.658
C08542=1049.685,146.409,411.691,171.060,35.424,156.657
C08543=1049.679,146.160,411.712,171.058,35.422,156.657
C08544=1049.673,145.911,411.733,171.056,35.420,156.656
C08545=1049.667,145.662,411.756,171.055,35.418,156.656
C08546=1049.661,145.413,411.777,171.053,35.416,156.656
C08547=1049.655,145.164,411.799,171.051,35.414,156.655
C08548=1049.649,144.916,411.820,171.049,35.412,156.655
C08549=1049.643,144.666,411.842,171.046,35.410,156.655
C08550=1049.636,144.417,411.863,171.044,35.408,156.654
C08551=1049.630,144.168,411.885,171.043,35.406,156.654
C08552=1049.624,143.920,411.906,171.041,35.404,156.653
C08553=1049.618,143.671,411.928,171.039,35.402,156.653
C08554=1049.612,143.421,411.949,171.037,35.400,156.653
C08555=1049.606,143.172,411.971,171.034,35.398,156.652
C08556=1049.600,142.924,411.992,171.033,35.396,156.652
C08557=1049.594,142.674,412.014,171.031,35.394,156.651
C08558=1049.588,142.425,412.035,171.029,35.392,156.651
C08559=1049.582,142.140,412.060,171.027,35.390,156.651
C08560=1049.574,141.855,412.084,171.025,35.388,156.650
C08561=1049.567,141.568,412.109,171.022,35.385,156.650
C08562=1049.561,141.283,412.134,171.020,35.383,156.650
C08563=1049.555,141.034,412.155,171.018,35.381,156.649
C08564=1049.548,140.786,412.176,171.016,35.379,156.649
C08565=1049.542,140.537,412.197,171.014,35.377,156.648
C08566=1049.536,140.287,412.219,171.013,35.375,156.648
C08567=1049.531,140.038,412.240,171.011,35.373,156.648
C08568=1049.525,139.789,412.261,171.008,35.371,156.647
C08569=1049.518,139.540,412.283,171.006,35.369,156.647
C08570=1049.513,139.291,412.304,171.004,35.367,156.647
C08571=1049.506,139.043,412.325,171.003,35.365,156.646
C08572=1049.500,138.793,412.347,171.001,35.363,156.646
C08573=1049.495,138.544,412.367,170.999,35.361,156.645
C08574=1049.488,138.295,412.389,170.996,35.359,156.645
C08575=1049.482,138.046,412.411,170.994,35.357,156.645
C08576=1049.476,137.798,412.431,170.993,35.355,156.644
C08577=1049.470,137.548,412.452,170.991,35.353,156.644
C08578=1049.464,137.299,412.474,170.989,35.351,156.644
C08579=1049.458,137.050,412.495,170.987,35.349,156.643
C08580=1049.451,136.801,412.516,170.986,35.347,156.643
C08581=1049.446,136.552,412.537,170.983,35.345,156.643
C08582=1049.440,136.303,412.558,170.981,35.344,156.642
C08583=1049.433,136.054,412.579,170.979,35.341,156.642
C08584=1049.428,135.805,412.601,170.978,35.339,156.641
C08585=1049.422,135.556,412.622,170.976,35.337,156.641
C08586=1049.415,135.307,412.643,170.974,35.335,156.641
C08587=1049.409,135.058,412.664,170.972,35.333,156.640
C08588=1049.403,134.808,412.685,170.969,35.332,156.640
C08589=1049.397,134.560,412.706,170.968,35.330,156.640
C08590=1049.391,134.311,412.727,170.966,35.328,156.639
C08591=1049.385,134.061,412.748,170.964,35.326,156.639
C08592=1049.379,133.813,412.769,170.962,35.323,156.639
C08593=1049.373,133.563,412.790,170.961,35.322,156.638
C08594=1049.367,133.315,412.811,170.959,35.320,156.638
C08595=1049.360,133.066,412.832,170.956,35.318,156.638
C08596=1049.355,132.817,412.853,170.954,35.316,156.637
C08597=1049.349,132.567,412.874,170.953,35.314,156.637
C08598=1049.342,132.318,412.895,170.951,35.312,156.637
C08599=1049.337,132.069,412.916,170.949,35.310,156.636
C08600=1049.331,131.820,412.937,170.947,35.308,156.636
C08601=1049.325,131.571,412.957,170.946,35.306,156.635
C08602=1049.319,131.322,412.979,170.943,35.304,156.635
C08603=1049.313,131.073,412.999,170.941,35.302,156.635
C08604=1049.307,130.823,413.020,170.939,35.300,156.634
C08605=1049.300,130.575,413.041,170.938,35.298,156.634
C08606=1049.295,130.325,413.062,170.936,35.296,156.634
C08607=1049.288,130.077,413.083,170.934,35.294,156.633
C08608=1049.282,129.828,413.103,170.932,35.293,156.633
C08609=1049.275,129.579,413.124,170.930,35.291,156.633
C08610=1049.269,129.329,413.144,170.928,35.289,156.632
C08611=1049.263,129.081,413.165,170.926,35.287,156.632
C08612=1049.257,128.831,413.186,170.924,35.285,156.632
C08613=1049.251,128.582,413.206,170.923,35.283,156.631
C08614=1049.245,128.333,413.228,170.921,35.281,156.631
C08615=1049.239,128.084,413.248,170.919,35.280,156.631
C08616=1049.232,127.835,413.269,170.917,35.278,156.630
C08617=1049.226,127.586,413.289,170.915,35.276,156.630
C08618=1049.220,127.337,413.310,170.913,35.274,156.630
C08619=1049.214,127.088,413.330,170.911,35.272,156.629
C08620=1049.208,126.839,413.351,170.909,35.270,156.629
C08621=1049.202,126.590,413.371,170.908,35.269,156.629
C08622=1049.195,126.341,413.392,170.906,35.267,156.628
C08623=1049.188,126.055,413.415,170.904,35.264,156.628
C08624=1049.181,125.770,413.439,170.901,35.262,156.627
C08625=1049.173,125.483,413.463,170.899,35.260,156.627
C08626=1049.166,125.198,413.486,170.897,35.258,156.627
C08627=1049.161,124.949,413.507,170.895,35.256,156.626
C08628=1049.155,124.699,413.527,170.893,35.254,156.626
C08629=1049.148,124.451,413.548,170.892,35.252,156.626
C08630=1049.142,124.201,413.569,170.890,35.250,156.625
C08631=1049.136,123.953,413.589,170.887,35.248,156.625
C08632=1049.130,123.704,413.609,170.886,35.246,156.625
C08633=1049.124,123.455,413.630,170.884,35.244,156.624
C08634=1049.118,123.206,413.650,170.882,35.243,156.624
C08635=1049.112,122.956,413.671,170.880,35.241,156.624
C08636=1049.106,122.707,413.691,170.879,35.239,156.623
C08637=1049.100,122.458,413.712,170.877,35.237,156.623
C08638=1049.094,122.209,413.732,170.875,35.235,156.623
C08639=1049.088,121.960,413.753,170.873,35.233,156.622
C08640=1049.082,121.711,413.773,170.871,35.231,156.622
C08641=1049.076,121.462,413.793,170.869,35.229,156.622
C08642=1049.070,121.212,413.814,170.868,35.227,156.621
C08643=1049.064,120.964,413.835,170.866,35.225,156.621
C08644=1049.057,120.714,413.855,170.864,35.224,156.620
C08645=1049.052,120.465,413.876,170.862,35.222,156.620
C08646=1049.046,120.216,413.896,170.860,35.220,156.620
C08647=1049.039,119.967,413.916,170.858,35.217,156.619
C08648=1049.033,119.718,413.936,170.856,35.215,156.619
C08649=1049.028,119.469,413.956,170.855,35.213,156.619
C08650=1049.021,119.220,413.977,170.853,35.212,156.618
C08651=1049.015,118.971,413.997,170.851,35.210,156.618
C08652=1049.010,118.722,414.018,170.850,35.208,156.618
C08653=1049.003,118.473,414.038,170.848,35.206,156.617
C08654=1048.997,118.224,414.058,170.845,35.204,156.617
C08655=1048.991,117.974,414.079,170.844,35.202,156.617
C08656=1048.985,117.725,414.099,170.842,35.200,156.616
C08657=1048.979,117.476,414.119,170.840,35.198,156.616
C08658=1048.973,117.228,414.139,170.838,35.196,156.616
C08659=1048.967,116.978,414.160,170.837,35.194,156.615
C08660=1048.961,116.729,414.180,170.835,35.193,156.615
C08661=1048.955,116.480,414.200,170.832,35.191,156.615
C08662=1048.949,116.231,414.220,170.831,35.189,156.614
C08663=1048.944,115.982,414.241,170.829,35.187,156.614
C08664=1048.938,115.733,414.261,170.827,35.185,156.614
C08665=1048.931,115.483,414.281,170.826,35.183,156.613
C08666=1048.926,115.234,414.302,170.824,35.181,156.613
C08667=1048.920,114.985,414.322,170.822,35.179,156.613
C08668=1048.914,114.736,414.341,170.821,35.177,156.612
C08669=1048.907,114.487,414.362,170.818,35.175,156.612
C08670=1048.902,114.238,414.382,170.816,35.173,156.611
C08671=1048.896,113.989,414.402,170.815,35.171,156.611
C08672=1048.889,113.739,414.423,170.813,35.169,156.611
C08673=1048.884,113.490,414.442,170.811,35.167,156.610
C08674=1048.878,113.241,414.462,170.810,35.165,156.610
C08675=1048.872,112.992,414.482,170.808,35.163,156.610
C08676=1048.865,112.743,414.502,170.806,35.162,156.609
C08677=1048.859,112.494,414.522,170.804,35.160,156.609
C08678=1048.853,112.245,414.542,170.802,35.158,156.609
C08679=1048.847,111.995,414.562,170.800,35.156,156.608
C08680=1048.841,111.746,414.582,170.799,35.155,156.608
C08681=1048.835,111.498,414.602,170.797,35.153,156.608
C08682=1048.829,111.249,414.622,170.795,35.151,156.607
C08683=1048.822,110.999,414.642,170.794,35.149,156.607
C08684=1048.816,110.750,414.661,170.792,35.147,156.607
C08685=1048.810,110.501,414.681,170.789,35.145,156.606
C08686=1048.804,110.251,414.701,170.788,35.143,156.606
C08687=1048.796,109.966,414.724,170.786,35.141,156.606
C08688=1048.790,109.680,414.747,170.784,35.139,156.605
C08689=1048.782,109.394,414.769,170.782,35.137,156.605
C08690=1048.776,109.108,414.792,170.780,35.135,156.605
C08691=1048.770,108.859,414.812,170.778,35.133,156.604
C08692=1048.764,108.610,414.832,170.776,35.131,156.604
C08693=1048.757,108.361,414.851,170.774,35.129,156.604
C08694=1048.751,108.112,414.871,170.772,35.127,156.603
C08695=1048.745,107.863,414.891,170.771,35.126,156.603
C08696=1048.739,107.613,414.910,170.769,35.124,156.603
C08697=1048.733,107.365,414.930,170.767,35.122,156.602
C08698=1048.727,107.116,414.950,170.766,35.120,156.602
C08699=1048.721,106.866,414.970,170.764,35.118,156.602
C08700=1048.714,106.617,414.989,170.762,35.116,156.601
C08701=1048.708,106.368,415.009,170.760,35.114,156.601
C08702=1048.702,106.119,415.028,170.758,35.113,156.601
C08703=1048.696,105.869,415.048,170.756,35.111,156.600
C08704=1048.690,105.620,415.068,170.755,35.109,156.600
C08705=1048.684,105.371,415.088,170.753,35.107,156.600
C08706=1048.677,105.123,415.107,170.751,35.106,156.599
C08707=1048.672,104.873,415.126,170.750,35.104,156.599
C08708=1048.665,104.624,415.147,170.748,35.102,156.599
C08709=1048.659,104.374,415.166,170.745,35.100,156.598
C08710=1048.653,104.126,415.186,170.744,35.098,156.598
C08711=1048.648,103.876,415.205,170.742,35.096,156.598
C08712=1048.641,103.628,415.224,170.740,35.094,156.597
C08713=1048.635,103.378,415.244,170.739,35.092,156.597
C08714=1048.629,103.129,415.264,170.737,35.090,156.597
C08715=1048.623,102.879,415.283,170.735,35.088,156.596
C08716=1048.617,102.630,415.303,170.734,35.087,156.596
C08717=1048.610,102.381,415.322,170.732,35.085,156.596
C08718=1048.604,102.132,415.342,170.730,35.083,156.595
C08719=1048.599,101.883,415.361,170.728,35.081,156.595
C08720=1048.593,101.634,415.381,170.726,35.079,156.595
C08721=1048.587,101.385,415.400,170.725,35.078,156.594
C08722=1048.580,101.136,415.420,170.723,35.076,156.594
C08723=1048.574,100.886,415.439,170.721,35.074,156.594
C08724=1048.568,100.637,415.459,170.720,35.072,156.593
C08725=1048.562,100.388,415.478,170.718,35.070,156.593
C08726=1048.556,100.139,415.497,170.715,35.068,156.593
C08727=1048.550,99.890,415.517,170.714,35.067,156.592
C08728=1048.544,99.641,415.536,170.712,35.065,156.592
C08729=1048.537,99.391,415.556,170.710,35.063,156.592
C08730=1048.531,99.142,415.575,170.709,35.061,156.591
C08731=1048.525,98.893,415.594,170.707,35.059,156.591
C08732=1048.519,98.644,415.614,170.705,35.058,156.591
C08733=1048.512,98.395,415.633,170.704,35.056,156.591
C08734=1048.507,98.145,415.652,170.702,35.054,156.590
C08735=1048.500,97.897,415.671,170.699,35.052,156.590
C08736=1048.494,97.647,415.690,170.698,35.050,156.590
C08737=1048.487,97.398,415.709,170.696,35.048,156.589
C08738=1048.482,97.148,415.729,170.695,35.047,156.589
C08739=1048.476,96.899,415.749,170.693,35.045,156.589
C08740=1048.469,96.650,415.767,170.691,35.043,156.588
C08741=1048.463,96.401,415.786,170.690,35.041,156.588
C08742=1048.457,96.152,415.806,170.688,35.039,156.588
C08743=1048.451,95.903,415.825,170.686,35.037,156.587
C08744=1048.445,95.654,415.844,170.684,35.036,156.587
C08745=1048.439,95.404,415.863,170.682,35.034,156.587
C08746=1048.433,95.155,415.882,170.680,35.032,156.586
C08747=1048.427,94.906,415.902,170.679,35.030,156.586
C08748=1048.420,94.657,415.920,170.677,35.028,156.586
C08749=1048.414,94.408,415.939,170.676,35.026,156.585
C08750=1048.408,94.159,415.958,170.674,35.025,156.585
C08751=1048.401,93.873,415.981,170.672,35.023,156.585
C08752=1048.394,93.586,416.003,170.669,35.021,156.584
C08753=1048.387,93.301,416.025,170.667,35.019,156.584
C08754=1048.380,93.015,416.046,170.665,35.016,156.584
C08755=1048.373,92.767,416.066,170.664,35.015,156.583
C08756=1048.368,92.517,416.085,170.662,35.013,156.583
C08757=1048.361,92.268,416.104,170.661,35.011,156.583
C08758=1048.356,92.019,416.123,170.659,35.009,156.582
C08759=1048.349,91.769,416.141,170.657,35.007,156.582
C08760=1048.344,91.520,416.161,170.656,35.005,156.582
C08761=1048.337,91.271,416.179,170.653,35.003,156.581
C08762=1048.331,91.021,416.199,170.651,35.002,156.581
C08763=1048.325,90.772,416.217,170.650,35.000,156.581
C08764=1048.319,90.524,416.237,170.648,34.998,156.580
C08765=1048.313,90.274,416.256,170.647,34.996,156.580
C08766=1048.307,90.025,416.275,170.645,34.994,156.580
C08767=1048.300,89.776,416.294,170.643,34.993,156.579
C08768=1048.294,89.527,416.312,170.642,34.991,156.579
C08769=1048.288,89.278,416.331,170.640,34.989,156.579
C08770=1048.282,89.028,416.350,170.637,34.987,156.579
C08771=1048.275,88.779,416.369,170.636,34.986,156.578
C08772=1048.269,88.530,416.388,170.634,34.984,156.578
C08773=1048.263,88.281,416.406,170.632,34.982,156.578
C08774=1048.257,88.031,416.425,170.631,34.980,156.577
C08775=1048.251,87.782,416.444,170.629,34.979,156.577
C08776=1048.244,87.533,416.463,170.627,34.977,156.577
C08777=1048.238,87.283,416.481,170.626,34.975,156.576
C08778=1048.232,87.034,416.500,170.624,34.973,156.576
C08779=1048.226,86.785,416.519,170.623,34.972,156.576
C08780=1048.219,86.536,416.537,170.620,34.970,156.576
C08781=1048.213,86.287,416.556,170.618,34.968,156.575
C08782=1048.207,86.037,416.575,170.617,34.966,156.575
C08783=1048.201,85.788,416.594,170.615,34.964,156.575
C08784=1048.194,85.539,416.612,170.613,34.963,156.574
C08785=1048.188,85.290,416.631,170.612,34.961,156.574
C08786=1048.182,85.040,416.650,170.610,34.959,156.574
C08787=1048.176,84.791,416.669,170.609,34.957,156.573
C08788=1048.170,84.542,416.687,170.607,34.956,156.573
C08789=1048.163,84.292,416.706,170.605,34.954,156.573
C08790=1048.158,84.044,416.724,170.603,34.952,156.572
C08791=1048.152,83.795,416.743,170.601,34.950,156.572
C08792=1048.145,83.545,416.762,170.599,34.948,156.572
C08793=1048.139,83.296,416.780,170.598,34.947,156.571
C08794=1048.133,83.047,416.798,170.596,34.945,156.571
C08795=1048.127,82.797,416.818,170.595,34.943,156.571
C08796=1048.121,82.548,416.836,170.593,34.941,156.570
C08797=1048.114,82.299,416.855,170.591,34.940,156.570
C08798=1048.108,82.050,416.873,170.590,34.938,156.570
C08799=1048.102,81.801,416.891,170.587,34.936,156.570
C08800=1048.097,81.551,416.910,170.585,34.934,156.569
C08801=1048.090,81.302,416.929,170.584,34.932,156.569
C08802=1048.084,81.053,416.948,170.582,34.931,156.569
C08803=1048.078,80.803,416.966,170.581,34.929,156.568
C08804=1048.071,80.554,416.984,170.579,34.927,156.568
C08805=1048.066,80.305,417.003,170.577,34.925,156.568
C08806=1048.060,80.056,417.022,170.576,34.923,156.567
C08807=1048.054,79.807,417.040,170.574,34.922,156.567
C08808=1048.047,79.557,417.058,170.572,34.920,156.567
C08809=1048.041,79.308,417.077,170.570,34.918,156.566
C08810=1048.035,79.059,417.095,170.568,34.916,156.566
C08811=1048.029,78.809,417.114,170.567,34.914,156.566
C08812=1048.023,78.561,417.132,170.565,34.913,156.566
C08813=1048.017,78.311,417.150,170.563,34.911,156.565
C08814=1048.011,78.062,417.169,170.562,34.909,156.565
C08815=1048.003,77.776,417.190,170.560,34.907,156.565
C08816=1047.996,77.490,417.211,170.558,34.905,156.564
C08817=1047.990,77.205,417.233,170.556,34.903,156.564
C08818=1047.982,76.919,417.254,170.553,34.901,156.563
C08819=1047.976,76.669,417.271,170.552,34.899,156.563
C08820=1047.970,76.420,417.290,170.550,34.897,156.563
C08821=1047.964,76.171,417.308,170.548,34.895,156.563
C08822=1047.957,75.922,417.326,170.547,34.894,156.562
C08823=1047.951,75.672,417.344,170.545,34.892,156.562
C08824=1047.945,75.423,417.363,170.544,34.890,156.562
C08825=1047.938,75.174,417.382,170.542,34.889,156.561
C08826=1047.933,74.925,417.399,170.540,34.887,156.561
C08827=1047.926,74.676,417.417,170.539,34.885,156.561
C08828=1047.920,74.426,417.435,170.537,34.883,156.560
C08829=1047.913,74.177,417.454,170.534,34.882,156.560
C08830=1047.907,73.927,417.472,170.533,34.880,156.560
C08831=1047.901,73.679,417.490,170.531,34.878,156.560
C08832=1047.895,73.429,417.508,170.530,34.877,156.559
C08833=1047.889,73.180,417.527,170.528,34.875,156.559
C08834=1047.883,72.930,417.545,170.526,34.873,156.559
C08835=1047.877,72.681,417.562,170.525,34.871,156.558
C08836=1047.871,72.432,417.581,170.523,34.870,156.558
C08837=1047.864,72.182,417.599,170.521,34.868,156.558
C08838=1047.858,71.933,417.617,170.520,34.866,156.557
C08839=1047.853,71.684,417.635,170.517,34.865,156.557
C08840=1047.845,71.435,417.653,170.516,34.863,156.557
C08841=1047.839,71.186,417.671,170.514,34.861,156.557
C08842=1047.833,70.936,417.690,170.512,34.859,156.556
C08843=1047.827,70.687,417.707,170.511,34.857,156.556
C08844=1047.821,70.438,417.725,170.509,34.856,156.556
C08845=1047.815,70.188,417.744,170.507,34.854,156.555
C08846=1047.809,69.939,417.762,170.506,34.852,156.555
C08847=1047.803,69.690,417.779,170.504,34.850,156.555
C08848=1047.796,69.441,417.797,170.503,34.848,156.554
C08849=1047.790,69.191,417.815,170.501,34.846,156.554
C08850=1047.784,68.941,417.833,170.498,34.845,156.554
C08851=1047.778,68.693,417.851,170.497,34.843,156.554
C08852=1047.771,68.444,417.869,170.495,34.841,156.553
C08853=1047.765,68.194,417.887,170.493,34.840,156.553
C08854=1047.759,67.945,417.905,170.492,34.838,156.553
C08855=1047.753,67.696,417.923,170.490,34.836,156.552
C08856=1047.746,67.446,417.940,170.489,34.835,156.552
C08857=1047.740,67.197,417.959,170.487,34.833,156.552
C08858=1047.734,66.948,417.976,170.485,34.831,156.552
C08859=1047.728,66.698,417.994,170.484,34.830,156.551
C08860=1047.721,66.449,418.012,170.482,34.828,156.551
C08861=1047.715,66.200,418.030,170.479,34.826,156.551
C08862=1047.709,65.951,418.048,170.478,34.824,156.550
C08863=1047.702,65.701,418.065,170.476,34.823,156.550
C08864=1047.697,65.452,418.083,170.474,34.821,156.550
C08865=1047.691,65.203,418.101,170.473,34.819,156.550
C08866=1047.684,64.953,418.119,170.471,34.817,156.549
C08867=1047.678,64.705,418.136,170.470,34.815,156.549
C08868=1047.672,64.455,418.154,170.468,34.814,156.549
C08869=1047.666,64.205,418.172,170.466,34.812,156.548
C08870=1047.659,63.956,418.190,170.465,34.810,156.548
C08871=1047.653,63.707,418.207,170.463,34.809,156.548
C08872=1047.647,63.457,418.224,170.460,34.807,156.547
C08873=1047.640,63.208,418.243,170.459,34.806,156.547
C08874=1047.634,62.959,418.260,170.457,34.804,156.547
C08875=1047.628,62.710,418.278,170.455,34.802,156.547
C08876=1047.621,62.460,418.295,170.454,34.801,156.546
C08877=1047.615,62.212,418.312,170.452,34.799,156.546
C08878=1047.609,61.962,418.330,170.450,34.797,156.546
C08879=1047.602,61.676,418.350,170.449,34.795,156.545
C08880=1047.594,61.389,418.371,170.447,34.793,156.545
C08881=1047.586,61.104,418.390,170.445,34.791,156.545
C08882=1047.579,60.818,418.411,170.443,34.790,156.545
C08883=1047.573,60.569,418.428,170.440,34.788,156.544
C08884=1047.566,60.319,418.446,170.439,34.786,156.544
C08885=1047.561,60.070,418.463,170.437,34.785,156.544
C08886=1047.554,59.821,418.481,170.435,34.783,156.543
C08887=1047.547,59.571,418.498,170.434,34.782,156.543
C08888=1047.541,59.322,418.516,170.432,34.780,156.543
C08889=1047.534,59.073,418.533,170.430,34.778,156.543
C08890=1047.529,58.824,418.551,170.429,34.776,156.542
C08891=1047.522,58.574,418.568,170.427,34.775,156.542
C08892=1047.516,58.324,418.585,170.425,34.773,156.542
C08893=1047.510,58.075,418.602,170.424,34.771,156.541
C08894=1047.503,57.826,418.619,170.422,34.770,156.541
C08895=1047.497,57.576,418.637,170.419,34.768,156.541
C08896=1047.491,57.327,418.654,170.418,34.767,156.541
C08897=1047.485,57.078,418.672,170.416,34.765,156.540
C08898=1047.478,56.829,418.689,170.414,34.763,156.540
C08899=1047.472,56.579,418.707,170.413,34.761,156.540
C08900=1047.466,56.330,418.724,170.411,34.760,156.540
C08901=1047.459,56.081,418.741,170.410,34.758,156.539
C08902=1047.453,55.831,418.759,170.408,34.756,156.539
C08903=1047.447,55.582,418.776,170.406,34.755,156.539
C08904=1047.440,55.332,418.793,170.405,34.753,156.538
C08905=1047.435,55.083,418.811,170.403,34.752,156.538
C08906=1047.428,54.834,418.828,170.401,34.750,156.538
C08907=1047.422,54.585,418.845,170.399,34.748,156.537
C08908=1047.415,54.335,418.863,170.397,34.746,156.537
C08909=1047.409,54.087,418.880,170.395,34.745,156.537
C08910=1047.403,53.836,418.897,170.394,34.743,156.537
C08911=1047.397,53.588,418.914,170.392,34.741,156.536
C08912=1047.390,53.338,418.931,170.390,34.740,156.536
C08913=1047.385,53.089,418.949,170.389,34.738,156.536
C08914=1047.378,52.840,418.966,170.387,34.736,156.536
C08915=1047.372,52.591,418.983,170.386,34.735,156.535
C08916=1047.366,52.341,419.000,170.384,34.733,156.535
C08917=1047.360,52.092,419.017,170.382,34.731,156.535
C08918=1047.353,51.842,419.035,170.381,34.730,156.534
C08919=1047.347,51.593,419.052,170.378,34.728,156.534
C08920=1047.341,51.343,419.069,170.376,34.726,156.534
C08921=1047.335,51.094,419.086,170.375,34.724,156.534
C08922=1047.328,50.845,419.104,170.373,34.723,156.533
C08923=1047.322,50.596,419.121,170.371,34.721,156.533
C08924=1047.316,50.346,419.138,170.370,34.719,156.533
C08925=1047.310,50.097,419.155,170.368,34.718,156.532
C08926=1047.303,49.848,419.172,170.366,34.716,156.532
C08927=1047.298,49.598,419.189,170.365,34.715,156.532
C08928=1047.291,49.349,419.206,170.363,34.713,156.532
C08929=1047.285,49.100,419.223,170.361,34.711,156.531
C08930=1047.280,48.850,419.240,170.360,34.709,156.531
C08931=1047.273,48.601,419.258,170.357,34.707,156.531
C08932=1047.266,48.352,419.275,170.356,34.705,156.530
C08933=1047.261,48.102,419.292,170.354,34.704,156.530
C08934=1047.254,47.853,419.309,170.352,34.702,156.530
C08935=1047.248,47.604,419.326,170.351,34.701,156.530
C08936=1047.242,47.354,419.343,170.349,34.699,156.529
C08937=1047.236,47.105,419.360,170.347,34.697,156.529
C08938=1047.229,46.856,419.377,170.346,34.696,156.529
C08939=1047.224,46.606,419.394,170.344,34.694,156.528
C08940=1047.218,46.357,419.411,170.342,34.692,156.528
C08941=1047.211,46.107,419.428,170.341,34.690,156.528
C08942=1047.206,45.858,419.445,170.339,34.689,156.528
C08943=1047.199,45.572,419.465,170.337,34.687,156.527
C08944=1047.191,45.285,419.484,170.334,34.685,156.527
C08945=1047.184,44.999,419.504,170.332,34.683,156.527
C08946=1047.177,44.713,419.523,170.331,34.681,156.526
C08947=1047.171,44.463,419.540,170.329,34.679,156.526
C08948=1047.165,44.214,419.558,170.327,34.677,156.526
C08949=1047.159,43.964,419.574,170.326,34.675,156.525
C08950=1047.153,43.716,419.591,170.324,34.674,156.525
C08951=1047.147,43.465,419.608,170.322,34.672,156.525
C08952=1047.141,43.217,419.625,170.321,34.670,156.525
C08953=1047.135,42.967,419.641,170.319,34.669,156.524
C08954=1047.128,42.718,419.659,170.317,34.667,156.524
C08955=1047.122,42.468,419.675,170.316,34.666,156.524
C08956=1047.115,42.219,419.692,170.313,34.664,156.523
C08957=1047.109,41.970,419.709,170.311,34.662,156.523
C08958=1047.103,41.720,419.725,170.310,34.660,156.523
C08959=1047.096,41.471,419.742,170.308,34.659,156.523
C08960=1047.090,41.222,419.758,170.306,34.657,156.522
C08961=1047.084,40.973,419.775,170.305,34.656,156.522
C08962=1047.078,40.723,419.792,170.303,34.654,156.522
C08963=1047.071,40.474,419.809,170.301,34.653,156.522
C08964=1047.065,40.225,419.825,170.300,34.651,156.521
C08965=1047.060,39.974,419.842,170.298,34.649,156.521
C08966=1047.053,39.726,419.859,170.296,34.647,156.521
C08967=1047.047,39.476,419.876,170.295,34.646,156.521
C08968=1047.041,39.226,419.892,170.293,34.644,156.520
C08969=1047.035,38.977,419.909,170.291,34.643,156.520
C08970=1047.029,38.728,419.925,170.289,34.641,156.520
C08971=1047.023,38.479,419.942,170.287,34.639,156.519
C08972=1047.016,38.229,419.959,170.285,34.637,156.519
C08973=1047.010,37.980,419.975,170.284,34.636,156.519
C08974=1047.004,37.731,419.992,170.282,34.634,156.519
C08975=1046.997,37.481,420.009,170.280,34.633,156.518
C08976=1046.991,37.232,420.025,170.279,34.631,156.518
C08977=1046.985,36.983,420.041,170.277,34.630,156.518
C08978=1046.978,36.733,420.057,170.275,34.628,156.518
C08979=1046.972,36.484,420.074,170.274,34.626,156.517
C08980=1046.966,36.235,420.091,170.272,34.625,156.517
C08981=1046.959,35.985,420.107,170.270,34.623,156.517
C08982=1046.953,35.735,420.124,170.268,34.622,156.517
C08983=1046.947,35.486,420.140,170.266,34.620,156.516
C08984=1046.941,35.237,420.157,170.264,34.618,156.516
C08985=1046.934,34.988,420.173,170.262,34.616,156.516
C08986=1046.928,34.738,420.189,170.261,34.615,156.515
C08987=1046.922,34.489,420.205,170.259,34.614,156.515
C08988=1046.915,34.239,420.222,170.257,34.612,156.515
C08989=1046.909,33.989,420.238,170.256,34.610,156.515
C08990=1046.903,33.741,420.255,170.254,34.609,156.514
C08991=1046.896,33.492,420.271,170.252,34.607,156.514
C08992=1046.890,33.242,420.287,170.250,34.605,156.514
C08993=1046.884,32.992,420.304,170.249,34.604,156.514
C08994=1046.878,32.743,420.320,170.247,34.603,156.513
C08995=1046.872,32.494,420.336,170.245,34.601,156.513
C08996=1046.865,32.244,420.352,170.244,34.599,156.513
C08997=1046.859,31.994,420.369,170.242,34.597,156.513
C08998=1046.852,31.746,420.386,170.239,34.596,156.512
C08999=1046.846,31.496,420.402,170.238,34.594,156.512
C09000=1046.840,31.247,420.418,170.236,34.593,156.512
C09001=1046.833,30.997,420.434,170.234,34.591,156.512
C09002=1046.827,30.748,420.450,170.233,34.589,156.511
C09003=1046.821,30.499,420.467,170.231,34.588,156.511
C09004=1046.815,30.249,420.483,170.229,34.586,156.511
C09005=1046.809,30.000,420.499,170.227,34.585,156.511
C09006=1046.802,29.750,420.515,170.226,34.583,156.510
C09007=1046.795,29.464,420.534,170.224,34.581,156.510
C09008=1046.789,29.178,420.553,170.222,34.579,156.510
C09009=1046.782,28.891,420.571,170.220,34.578,156.509
C09010=1046.774,28.605,420.589,170.218,34.576,156.509
C09011=1046.768,28.355,420.606,170.216,34.574,156.509
C09012=1046.762,28.106,420.622,170.213,34.572,156.509
C09013=1046.755,27.857,420.638,170.212,34.571,156.508
C09014=1046.749,27.607,420.654,170.210,34.570,156.508
C09015=1046.743,27.358,420.670,170.208,34.568,156.508
C09016=1046.736,27.109,420.686,170.207,34.566,156.508
C09017=1046.730,26.859,420.703,170.205,34.565,156.507
C09018=1046.724,26.609,420.719,170.203,34.563,156.507
C09019=1046.717,26.360,420.734,170.201,34.562,156.507
C09020=1046.712,26.110,420.750,170.200,34.560,156.507
C09021=1046.705,25.861,420.766,170.198,34.558,156.506
C09022=1046.699,25.612,420.782,170.196,34.557,156.506
C09023=1046.692,25.362,420.798,170.195,34.556,156.506
C09024=1046.686,25.113,420.814,170.193,34.554,156.506
C09025=1046.680,24.864,420.830,170.191,34.552,156.505
C09026=1046.673,24.615,420.846,170.189,34.551,156.505
C09027=1046.667,24.365,420.862,170.188,34.549,156.505
C09028=1046.661,24.116,420.877,170.186,34.548,156.505
C09029=1046.655,23.866,420.894,170.183,34.546,156.504
C09030=1046.647,23.616,420.910,170.181,34.544,156.504
C09031=1046.641,23.367,420.926,170.180,34.543,156.504
C09032=1046.636,23.118,420.942,170.178,34.542,156.504
C09033=1046.629,22.868,420.957,170.176,34.540,156.503
C09034=1046.623,22.619,420.973,170.175,34.538,156.503
C09035=1046.617,22.370,420.989,170.173,34.537,156.503
C09036=1046.611,22.120,421.005,170.171,34.535,156.503
C09037=1046.604,21.871,421.020,170.169,34.534,156.502
C09038=1046.598,21.621,421.036,170.168,34.532,156.502
C09039=1046.592,21.372,421.052,170.166,34.530,156.502
C09040=1046.586,21.123,421.068,170.164,34.529,156.502
C09041=1046.579,20.872,421.084,170.162,34.528,156.501
C09042=1046.573,20.623,421.100,170.161,34.526,156.501
C09043=1046.567,20.374,421.116,170.159,34.524,156.501
C09044=1046.560,20.125,421.132,170.157,34.523,156.501
C09045=1046.554,19.875,421.147,170.154,34.521,156.500
C09046=1046.548,19.626,421.163,170.153,34.520,156.500
C09047=1046.542,19.376,421.179,170.151,34.518,156.500
C09048=1046.535,19.127,421.194,170.149,34.517,156.500
C09049=1046.529,18.878,421.210,170.147,34.515,156.499
C09050=1046.523,18.628,421.225,170.146,34.514,156.499
C09051=1046.516,18.379,421.241,170.144,34.512,156.499
C09052=1046.510,18.129,421.257,170.142,34.511,156.499
C09053=1046.504,17.880,421.272,170.140,34.509,156.498
C09054=1046.497,17.631,421.288,170.139,34.508,156.498
C09055=1046.491,17.381,421.304,170.137,34.506,156.498
C09056=1046.485,17.132,421.319,170.135,34.505,156.498
C09057=1046.479,16.882,421.335,170.133,34.503,156.497
C09058=1046.473,16.633,421.350,170.132,34.502,156.497
C09059=1046.466,16.384,421.366,170.130,34.500,156.497
C09060=1046.460,16.134,421.382,170.128,34.499,156.497
C09061=1046.454,15.885,421.397,170.126,34.497,156.497
C09062=1046.448,15.635,421.413,170.124,34.495,156.496
C09063=1046.441,15.386,421.428,170.122,34.494,156.496
C09064=1046.435,15.137,421.444,170.120,34.493,156.496
C09065=1046.429,14.887,421.460,170.118,34.491,156.496
C09066=1046.422,14.638,421.475,170.117,34.489,156.495
C09067=1046.417,14.388,421.491,170.115,34.488,156.495
C09068=1046.410,14.139,421.507,170.113,34.486,156.495
C09069=1046.404,13.889,421.521,170.111,34.485,156.495
C09070=1046.397,13.640,421.537,170.110,34.484,156.494
C09071=1046.390,13.354,421.554,170.107,34.482,156.494
C09072=1046.382,13.069,421.572,170.105,34.480,156.494
C09073=1046.375,12.784,421.589,170.103,34.478,156.494
C09074=1046.368,12.499,421.607,170.101,34.477,156.493
C09075=1046.362,12.250,421.623,170.100,34.476,156.493
C09076=1046.355,12.000,421.638,170.098,34.474,156.493
C09077=1046.349,11.751,421.653,170.096,34.472,156.493
C09078=1046.342,11.501,421.669,170.094,34.471,156.492
C09079=1046.336,11.252,421.684,170.092,34.470,156.492
C09080=1046.329,11.003,421.699,170.091,34.468,156.492
C09081=1046.323,10.753,421.714,170.088,34.467,156.492
C09082=1046.317,10.503,421.730,170.086,34.466,156.492
C09083=1046.310,10.254,421.745,170.084,34.464,156.491
C09084=1046.304,10.004,421.760,170.082,34.462,156.491
C09085=1046.298,9.755,421.775,170.081,34.461,156.491
C09086=1046.291,9.506,421.791,170.079,34.460,156.491
C09087=1046.285,9.256,421.806,170.077,34.458,156.490
C09088=1046.278,9.006,421.821,170.075,34.457,156.490
C09089=1046.272,8.757,421.837,170.073,34.456,156.490
C09090=1046.266,8.507,421.852,170.072,34.454,156.490
C09091=1046.259,8.258,421.867,170.070,34.452,156.490
C09092=1046.253,8.008,421.882,170.068,34.451,156.489
C09093=1046.246,7.759,421.898,170.066,34.450,156.489
C09094=1046.241,7.510,421.912,170.064,34.448,156.489
C09095=1046.234,7.260,421.927,170.063,34.447,156.489
C09096=1046.228,7.011,421.942,170.061,34.446,156.488
C09097=1046.221,6.762,421.958,170.059,34.444,156.488
C09098=1046.216,6.512,421.973,170.057,34.442,156.488
C09099=1046.209,6.262,421.988,170.055,34.441,156.488
C09100=1046.203,6.013,422.003,170.054,34.440,156.488
C09101=1046.196,5.763,422.019,170.051,34.438,156.487
C09102=1046.190,5.515,422.033,170.049,34.437,156.487
C09103=1046.184,5.265,422.048,170.047,34.435,156.487
C09104=1046.177,5.015,422.063,170.045,34.433,156.487
